# B&R Automation Studio project reAM250plc (part 2)

#### IOModule_X20AI4622.cpp
```cpp
/*++

Copyright (C) 2024 Institute for Machine Tools and Industrial Management
TUM School of Engineering and Design
Technical University of Munich

All rights reserved.

Redistribution and use in source and binary forms, with or without
modification, are permitted provided that the following conditions are met:
	* Redistributions of source code must retain the above copyright
	  notice, this list of conditions and the following disclaimer.
	* Redistributions in binary form must reproduce the above copyright
	  notice, this list of conditions and the following disclaimer in the
	  documentation and/or other materials provided with the distribution.
	* Neither the name of the Technical University of Munich nor the
	  names of its contributors may be used to endorse or promote products
	  derived from this software without specific prior written permission.

THIS SOFTWARE IS PROVIDED BY THE COPYRIGHT HOLDERS AND CONTRIBUTORS "AS IS" AND
ANY EXPRESS OR IMPLIED WARRANTIES, INCLUDING, BUT NOT LIMITED TO, THE IMPLIED
WARRANTIES OF MERCHANTABILITY AND FITNESS FOR A PARTICULAR PURPOSE ARE
DISCLAIMED. IN NO EVENT SHALL TECHNICAL UNIVERSITY OF MUNICH BE LIABLE FOR ANY
DIRECT, INDIRECT, INCIDENTAL, SPECIAL, EXEMPLARY, OR CONSEQUENTIAL DAMAGES
(INCLUDING, BUT NOT LIMITED TO, PROCUREMENT OF SUBSTITUTE GOODS OR SERVICES;
LOSS OF USE, DATA, OR PROFITS; OR BUSINESS INTERRUPTION) HOWEVER CAUSED AND
ON ANY THEORY OF LIABILITY, WHETHER IN CONTRACT, STRICT LIABILITY, OR TORT
(INCLUDING NEGLIGENCE OR OTHERWISE) ARISING IN ANY WAY OUT OF THE USE OF THIS
SOFTWARE, EVEN IF ADVISED OF THE POSSIBILITY OF SUCH DAMAGE.

*/

#include "IOModule_X20AI4622.hpp"

// Raw Registers
#define JOURNALVARIABLE_X20AI4622_MODULEOK 1
#define JOURNALVARIABLE_X20AI4622_STALEDATA 2
#define JOURNALVARIABLE_X20AI4622_SERIALNUMBER 3
#define JOURNALVARIABLE_X20AI4622_MODULEID 4
#define JOURNALVARIABLE_X20AI4622_HARDWAREVARIANT 5
#define JOURNALVARIABLE_X20AI4622_FIRMWAREVERSION 6
#define JOURNALVARIABLE_X20AI4622_ANALOGINPUT01 7
#define JOURNALVARIABLE_X20AI4622_ANALOGINPUT02 8
#define JOURNALVARIABLE_X20AI4622_ANALOGINPUT03 9
#define JOURNALVARIABLE_X20AI4622_ANALOGINPUT04 10
#define JOURNALVARIABLE_X20AI4622_STATUSINPUT01 11

// Derived Values
#define JOURNALVARIABLE_X20AI4622_INPUTVOLTAGE01 1001
#define JOURNALVARIABLE_X20AI4622_INPUTVOLTAGE02 1002
#define JOURNALVARIABLE_X20AI4622_INPUTVOLTAGE03 1003
#define JOURNALVARIABLE_X20AI4622_INPUTVOLTAGE04 1004
#define JOURNALVARIABLE_X20AI4622_INPUTCURRENTINAMPERE01 1005
#define JOURNALVARIABLE_X20AI4622_INPUTCURRENTINAMPERE02 1006
#define JOURNALVARIABLE_X20AI4622_INPUTCURRENTINAMPERE03 1007
#define JOURNALVARIABLE_X20AI4622_INPUTCURRENTINAMPERE04 1008

namespace BuRCPP {

	CIOModule_X20AI4622	::CIOModule_X20AI4622 (const std::string & sName, IOMappingX20AI4622_TYP * pMapping)
	: CIOModule (sName), m_pMapping (pMapping)
	{
		for (auto &channelType:m_ChannelTypes)
			channelType = eIOChannelType_X20AI4622::mtVoltage10V;

		for (auto &LowerLimits:m_nLowerLimit)
			LowerLimits = -32767;

		for (auto &UpperLimits:m_nUpperLimit)
			UpperLimits = 32766;

	}

	CIOModule_X20AI4622::~CIOModule_X20AI4622 ()
	{

	}

	void CIOModule_X20AI4622::onRegisterJournal ()
	{
		registerBoolValue ("ModuleOk", JOURNALVARIABLE_X20AI4622_MODULEOK);
		registerBoolValue ("StaleData", JOURNALVARIABLE_X20AI4622_STALEDATA);
		registerUInt32Value ("SerialNumber", JOURNALVARIABLE_X20AI4622_SERIALNUMBER);
		registerUInt16Value ("ModuleID", JOURNALVARIABLE_X20AI4622_MODULEID);
		registerUInt16Value ("HardwareVariant", JOURNALVARIABLE_X20AI4622_HARDWAREVARIANT);
		registerUInt16Value ("FirmwareVersion", JOURNALVARIABLE_X20AI4622_FIRMWAREVERSION);
		registerInt16Value ("AnalogInput01", JOURNALVARIABLE_X20AI4622_ANALOGINPUT01);
		registerInt16Value ("AnalogInput02", JOURNALVARIABLE_X20AI4622_ANALOGINPUT02);
		registerInt16Value ("AnalogInput03", JOURNALVARIABLE_X20AI4622_ANALOGINPUT03);
		registerInt16Value ("AnalogInput04", JOURNALVARIABLE_X20AI4622_ANALOGINPUT04);
		registerUInt8Value ("StatusInput01", JOURNALVARIABLE_X20AI4622_STATUSINPUT01);

		switch (getChannelType (1)) {
			case eIOChannelType_X20AI4622::mtVoltage10V:
				registerDoubleValue ("InputVoltage01", JOURNALVARIABLE_X20AI4622_INPUTVOLTAGE01, -10.0, 10.0, 65536);
				break;

			case eIOChannelType_X20AI4622::mtCurrent0to20mA:
				registerDoubleValue ("InputCurrentInAmpere01", JOURNALVARIABLE_X20AI4622_INPUTCURRENTINAMPERE01, 0.000, 0.020, 65536);
				break;

			case eIOChannelType_X20AI4622::mtCurrent4to20mA:
				registerDoubleValue ("InputCurrentInAmpere01", JOURNALVARIABLE_X20AI4622_INPUTCURRENTINAMPERE01, 0.004, 0.020, 65536);
				break;
		}

		switch (getChannelType (2)) {
			case eIOChannelType_X20AI4622::mtVoltage10V:
				registerDoubleValue ("InputVoltage02", JOURNALVARIABLE_X20AI4622_INPUTVOLTAGE02, -10.0, 10.0, 65536);
				break;

			case eIOChannelType_X20AI4622::mtCurrent0to20mA:
				registerDoubleValue ("InputCurrentInAmpere02", JOURNALVARIABLE_X20AI4622_INPUTCURRENTINAMPERE02, 0.000, 0.020, 65536);
				break;

			case eIOChannelType_X20AI4622::mtCurrent4to20mA:
				registerDoubleValue ("InputCurrentInAmpere02", JOURNALVARIABLE_X20AI4622_INPUTCURRENTINAMPERE02, 0.004, 0.020, 65536);
				break;
		}

		switch (getChannelType (3)) {
			case eIOChannelType_X20AI4622::mtVoltage10V:
				registerDoubleValue ("InputVoltage03", JOURNALVARIABLE_X20AI4622_INPUTVOLTAGE03, -10.0, 10.0, 65536);
				break;

			case eIOChannelType_X20AI4622::mtCurrent0to20mA:
				registerDoubleValue ("InputCurrentInAmpere03", JOURNALVARIABLE_X20AI4622_INPUTCURRENTINAMPERE03, 0.000, 0.020, 65536);
				break;

			case eIOChannelType_X20AI4622::mtCurrent4to20mA:
				registerDoubleValue ("InputCurrentInAmpere03", JOURNALVARIABLE_X20AI4622_INPUTCURRENTINAMPERE03, 0.004, 0.020, 65536);
				break;
		}

		switch (getChannelType (4)) {
			case eIOChannelType_X20AI4622::mtVoltage10V:
				registerDoubleValue ("InputVoltage04", JOURNALVARIABLE_X20AI4622_INPUTVOLTAGE04, -10.0, 10.0, 65536);
				break;

			case eIOChannelType_X20AI4622::mtCurrent0to20mA:
				registerDoubleValue ("InputCurrentInAmpere04", JOURNALVARIABLE_X20AI4622_INPUTCURRENTINAMPERE04, 0.000, 0.020, 65536);
				break;

			case eIOChannelType_X20AI4622::mtCurrent4to20mA:
				registerDoubleValue ("InputCurrentInAmpere04", JOURNALVARIABLE_X20AI4622_INPUTCURRENTINAMPERE04, 0.004, 0.020, 65536);
				break;
		}
	}

	void CIOModule_X20AI4622::onUpdateJournal ()
	{
		setBoolValue (JOURNALVARIABLE_X20AI4622_MODULEOK, m_pMapping->ModuleOk);
		setBoolValue (JOURNALVARIABLE_X20AI4622_STALEDATA, m_pMapping->StaleData);
		setIntegerValue (JOURNALVARIABLE_X20AI4622_SERIALNUMBER, m_pMapping->SerialNumber);
		setIntegerValue (JOURNALVARIABLE_X20AI4622_MODULEID, m_pMapping->ModuleID);
		setIntegerValue (JOURNALVARIABLE_X20AI4622_HARDWAREVARIANT, m_pMapping->HardwareVariant);
		setIntegerValue (JOURNALVARIABLE_X20AI4622_FIRMWAREVERSION, m_pMapping->FirmwareVersion);
		setIntegerValue (JOURNALVARIABLE_X20AI4622_ANALOGINPUT01, m_pMapping->AnalogInput01);
		setIntegerValue (JOURNALVARIABLE_X20AI4622_ANALOGINPUT02, m_pMapping->AnalogInput02);
		setIntegerValue (JOURNALVARIABLE_X20AI4622_ANALOGINPUT03, m_pMapping->AnalogInput03);
		setIntegerValue (JOURNALVARIABLE_X20AI4622_ANALOGINPUT04, m_pMapping->AnalogInput04);
		setIntegerValue (JOURNALVARIABLE_X20AI4622_STATUSINPUT01, m_pMapping->StatusInput01);

		for (int index = 0; index < 4; index++)
		{
			uint32_t nChannelNo = index + 1;
			switch (getChannelType (nChannelNo)) {

				case eIOChannelType_X20AI4622::mtVoltage10V:

					setDoubleValue (JOURNALVARIABLE_X20AI4622_INPUTVOLTAGE01 + index, getInputVoltageInVolt (nChannelNo));
					/*setDoubleValue (JOURNALVARIABLE_X20AI4622_INPUTVOLTAGE02, getInputVoltageInVolt (2));
					setDoubleValue (JOURNALVARIABLE_X20AI4622_INPUTVOLTAGE03, getInputVoltageInVolt (3));
					setDoubleValue (JOURNALVARIABLE_X20AI4622_INPUTVOLTAGE04, getInputVoltageInVolt (4));*/
					break;

				case eIOChannelType_X20AI4622::mtCurrent0to20mA:
				case eIOChannelType_X20AI4622::mtCurrent4to20mA:
					setDoubleValue (JOURNALVARIABLE_X20AI4622_INPUTCURRENTINAMPERE01 + index, getInputCurrentInAmpere (nChannelNo));
					/*setDoubleValue (JOURNALVARIABLE_X20AI4622_INPUTCURRENTINAMPERE02, getInputCurrentInAmpere (2));
					setDoubleValue (JOURNALVARIABLE_X20AI4622_INPUTCURRENTINAMPERE03, getInputCurrentInAmpere (3));
					setDoubleValue (JOURNALVARIABLE_X20AI4622_INPUTCURRENTINAMPERE04, getInputCurrentInAmpere (4));*/
					break;
			}
		}
	}

	bool CIOModule_X20AI4622::isActive ()
	{
		return m_pMapping->ModuleOk != 0;
	}

	uint32_t CIOModule_X20AI4622::getSerialNumber ()
	{
		return m_pMapping->SerialNumber;
	}

	uint16_t CIOModule_X20AI4622::getModuleID ()
	{
		return m_pMapping->ModuleID;
	}

	uint16_t CIOModule_X20AI4622::getHardwareVariant ()
	{
		return m_pMapping->HardwareVariant;
	}

	uint16_t CIOModule_X20AI4622::getFirmwareVersion ()
	{
		return m_pMapping->FirmwareVersion;
	}

	int16_t CIOModule_X20AI4622::getRawValue (uint32_t nChannelNo)
	{

		switch (nChannelNo) {
			case 1: return m_pMapping->AnalogInput01;
			case 2: return m_pMapping->AnalogInput02;
			case 3: return m_pMapping->AnalogInput03;
			case 4: return m_pMapping->AnalogInput04;
			default:
				throw CException (eErrorCode::INVALIDCHANNELNUMBER, "invalid channel number: " + std::to_string (nChannelNo));
		}
	}

	double CIOModule_X20AI4622::getRawValueNormalizedZeroToOne (uint32_t nChannelNo)
	{
		if (nChannelNo > 0 && nChannelNo < 5)
		{
			int32_t rawValue = getRawValue (nChannelNo);
			int32_t nRange = m_nUpperLimit[nChannelNo -1] - m_nLowerLimit[nChannelNo -1];
			return (double) (rawValue - (int32_t) m_nLowerLimit[nChannelNo -1]) / (double) nRange;
		}
		else
		{
			throw CException (eErrorCode::INVALIDCHANNELNUMBER, "invalid channel number: " + std::to_string (nChannelNo));
		}
	}

	double CIOModule_X20AI4622::getInputVoltageInVolt (uint32_t nChannelNo)
	{
		switch (getChannelType (nChannelNo)) {
			case eIOChannelType_X20AI4622::mtVoltage10V:
				return (getRawValueNormalizedZeroToOne (nChannelNo) - 0.5) * 20.0;
			default:
				throw CException (eErrorCode::NOVOLTAGEMODULE, "IO module does not measure voltage: " + m_sName );
		}

	}

	double CIOModule_X20AI4622::getInputCurrentInAmpere (uint32_t nChannelNo)
	{
		switch (getChannelType (nChannelNo)) {
			case eIOChannelType_X20AI4622::mtCurrent0to20mA:
				return (getRawValueNormalizedZeroToOne (nChannelNo)) * 0.020;
			case eIOChannelType_X20AI4622::mtCurrent4to20mA:
				return (getRawValueNormalizedZeroToOne (nChannelNo)) * 0.016 + 0.004;
			default:
				throw CException (eErrorCode::NOCURRENTMODULE, "IO module does not measure current: " + m_sName );
		}

	}

	bool CIOModule_X20AI4622::setRange(uint32_t nChannelNo, uint16_t nLower, uint16_t nUpper)
	{
		if (nChannelNo > 0 && nChannelNo < 5)
		{
			m_nLowerLimit[nChannelNo - 1] = nLower;
			m_nUpperLimit[nChannelNo - 1] = nUpper;
			return true;
		}
		else
		{
			return false;
		}
	}

	uint16_t CIOModule_X20AI4622::getIOStatus (uint32_t nChannelNo)
	{
		//status IDs: 0 = no error, 1 = lower limit value undershot, 2 = upper limit value exceeded, 3 = wire breakage
		switch (nChannelNo) {
			case 1: return (m_pMapping->StatusInput01 & 0x03);
			case 2: return ((m_pMapping->StatusInput01 >> 2) & 0x03);
			case 3: return ((m_pMapping->StatusInput01 >> 4) & 0x03);
			case 4: return ((m_pMapping->StatusInput01 >> 6) & 0x03);
			default:
				throw CException (eErrorCode::INVALIDCHANNELNUMBER, "invalid channel number: " + std::to_string (nChannelNo));
		}
	}

	eIOChannelType_X20AI4622 CIOModule_X20AI4622::getChannelType (uint32_t nChannelNo)
	{
		if ((nChannelNo >= 1) && (nChannelNo <= 4))
		{
			return m_ChannelTypes[nChannelNo - 1];
		}
		else
			return eIOChannelType_X20AI4622::mtUnknown;
	}

	bool CIOModule_X20AI4622::setChannelType (uint32_t nChannelNo, eIOChannelType_X20AI4622 eChannelTypes)
	{
		if ((nChannelNo >= 1) && (nChannelNo <= 4))
		{
			switch (eChannelTypes) {
				case eIOChannelType_X20AI4622::mtVoltage10V:
					setRange(nChannelNo, -32768 , 32767);
					break;
				case eIOChannelType_X20AI4622::mtCurrent0to20mA:
					setRange(nChannelNo, 0, 32767);
					break;
				case eIOChannelType_X20AI4622::mtCurrent4to20mA:
					setRange(nChannelNo, -8192 , 32767);
					break;
				default:
					throw CException (eErrorCode::INVALIDCHANNELTYPE, "invalid channel type");
			}
			m_ChannelTypes[nChannelNo - 1] = eChannelTypes;
			return true;
		}
		else
		{
			throw CException (eErrorCode::INVALIDCHANNELNUMBER, "invalid channel number: " + std::to_string (nChannelNo));
		}
	}

}
```

#### IOModule_X20DI6371.hpp
```cpp
/*++

Copyright (C) 2024 Institute for Machine Tools and Industrial Management
TUM School of Engineering and Design
Technical University of Munich

All rights reserved.

Redistribution and use in source and binary forms, with or without
modification, are permitted provided that the following conditions are met:
	* Redistributions of source code must retain the above copyright
	  notice, this list of conditions and the following disclaimer.
	* Redistributions in binary form must reproduce the above copyright
	  notice, this list of conditions and the following disclaimer in the
	  documentation and/or other materials provided with the distribution.
	* Neither the name of the Technical University of Munich nor the
	  names of its contributors may be used to endorse or promote products
	  derived from this software without specific prior written permission.

THIS SOFTWARE IS PROVIDED BY THE COPYRIGHT HOLDERS AND CONTRIBUTORS "AS IS" AND
ANY EXPRESS OR IMPLIED WARRANTIES, INCLUDING, BUT NOT LIMITED TO, THE IMPLIED
WARRANTIES OF MERCHANTABILITY AND FITNESS FOR A PARTICULAR PURPOSE ARE
DISCLAIMED. IN NO EVENT SHALL TECHNICAL UNIVERSITY OF MUNICH BE LIABLE FOR ANY
DIRECT, INDIRECT, INCIDENTAL, SPECIAL, EXEMPLARY, OR CONSEQUENTIAL DAMAGES
(INCLUDING, BUT NOT LIMITED TO, PROCUREMENT OF SUBSTITUTE GOODS OR SERVICES;
LOSS OF USE, DATA, OR PROFITS; OR BUSINESS INTERRUPTION) HOWEVER CAUSED AND
ON ANY THEORY OF LIABILITY, WHETHER IN CONTRACT, STRICT LIABILITY, OR TORT
(INCLUDING NEGLIGENCE OR OTHERWISE) ARISING IN ANY WAY OUT OF THE USE OF THIS
SOFTWARE, EVEN IF ADVISED OF THE POSSIBILITY OF SUCH DAMAGE.

*/

#ifndef __IOMODULE_X20DI6371_HPP
#define __IOMODULE_X20DI6371_HPP

#include "../Framework/Framework.hpp"

namespace BuRCPP {

	class CIOModule_X20DI6371 : public CIOModule {
		protected:
		IOMappingX20DI6371_TYP * m_pMapping;

		public:
		CIOModule_X20DI6371 (const std::string & sName, IOMappingX20DI6371_TYP * pMapping);
		virtual ~CIOModule_X20DI6371 ();

		bool isActive () override;
		uint32_t getSerialNumber () override;
		uint16_t getModuleID () override;
		uint16_t getHardwareVariant () override;
		uint16_t getFirmwareVersion () override;

		uint16_t getInput (uint32_t);

		void onRegisterJournal ();
		void onUpdateJournal ();

	};

}

#endif // __IOMODULE_X20DI6371_HPP
```

#### IOModule_X20DI6371.cpp
```cpp
/*++

Copyright (C) 2024 Institute for Machine Tools and Industrial Management
TUM School of Engineering and Design
Technical University of Munich

All rights reserved.

Redistribution and use in source and binary forms, with or without
modification, are permitted provided that the following conditions are met:
	* Redistributions of source code must retain the above copyright
	  notice, this list of conditions and the following disclaimer.
	* Redistributions in binary form must reproduce the above copyright
	  notice, this list of conditions and the following disclaimer in the
	  documentation and/or other materials provided with the distribution.
	* Neither the name of the Technical University of Munich nor the
	  names of its contributors may be used to endorse or promote products
	  derived from this software without specific prior written permission.

THIS SOFTWARE IS PROVIDED BY THE COPYRIGHT HOLDERS AND CONTRIBUTORS "AS IS" AND
ANY EXPRESS OR IMPLIED WARRANTIES, INCLUDING, BUT NOT LIMITED TO, THE IMPLIED
WARRANTIES OF MERCHANTABILITY AND FITNESS FOR A PARTICULAR PURPOSE ARE
DISCLAIMED. IN NO EVENT SHALL TECHNICAL UNIVERSITY OF MUNICH BE LIABLE FOR ANY
DIRECT, INDIRECT, INCIDENTAL, SPECIAL, EXEMPLARY, OR CONSEQUENTIAL DAMAGES
(INCLUDING, BUT NOT LIMITED TO, PROCUREMENT OF SUBSTITUTE GOODS OR SERVICES;
LOSS OF USE, DATA, OR PROFITS; OR BUSINESS INTERRUPTION) HOWEVER CAUSED AND
ON ANY THEORY OF LIABILITY, WHETHER IN CONTRACT, STRICT LIABILITY, OR TORT
(INCLUDING NEGLIGENCE OR OTHERWISE) ARISING IN ANY WAY OUT OF THE USE OF THIS
SOFTWARE, EVEN IF ADVISED OF THE POSSIBILITY OF SUCH DAMAGE.

*/

#include "IOModule_X20DI6371.hpp"

// Raw Registers
#define JOURNALVARIABLE_X20DI6371_MODULEOK 1
#define JOURNALVARIABLE_X20DI6371_SERIALNUMBER 2
#define JOURNALVARIABLE_X20DI6371_MODULEID 3
#define JOURNALVARIABLE_X20DI6371_HARDWAREVARIANT 4
#define JOURNALVARIABLE_X20DI6371_FIRMWAREVERSION 5
#define JOURNALVARIABLE_X20DI6371_DIGITALINPUT01 6
#define JOURNALVARIABLE_X20DI6371_DIGITALINPUT02 7
#define JOURNALVARIABLE_X20DI6371_DIGITALINPUT03 8
#define JOURNALVARIABLE_X20DI6371_DIGITALINPUT04 9
#define JOURNALVARIABLE_X20DI6371_DIGITALINPUT05 10
#define JOURNALVARIABLE_X20DI6371_DIGITALINPUT06 11

namespace BuRCPP {

	CIOModule_X20DI6371::CIOModule_X20DI6371 (const std::string & sName, IOMappingX20DI6371_TYP * pMapping)
		: CIOModule (sName), m_pMapping (pMapping)
	{

	}

	CIOModule_X20DI6371::~CIOModule_X20DI6371 ()
	{
	}

	void CIOModule_X20DI6371::onRegisterJournal ()
	{
		registerBoolValue ("ModuleOk", JOURNALVARIABLE_X20DI6371_MODULEOK);
		registerUInt32Value ("SerialNumber", JOURNALVARIABLE_X20DI6371_SERIALNUMBER);
		registerUInt16Value ("ModuleID", JOURNALVARIABLE_X20DI6371_MODULEID);
		registerUInt16Value ("HardwareVariant", JOURNALVARIABLE_X20DI6371_HARDWAREVARIANT);
		registerUInt16Value ("FirmwareVersion", JOURNALVARIABLE_X20DI6371_FIRMWAREVERSION);
		registerBoolValue ("DigitalInput01", JOURNALVARIABLE_X20DI6371_DIGITALINPUT01);
		registerBoolValue ("DigitalInput02", JOURNALVARIABLE_X20DI6371_DIGITALINPUT02);
		registerBoolValue ("DigitalInput03", JOURNALVARIABLE_X20DI6371_DIGITALINPUT03);
		registerBoolValue ("DigitalInput04", JOURNALVARIABLE_X20DI6371_DIGITALINPUT04);
		registerBoolValue ("DigitalInput05", JOURNALVARIABLE_X20DI6371_DIGITALINPUT05);
		registerBoolValue ("DigitalInput06", JOURNALVARIABLE_X20DI6371_DIGITALINPUT06);

	}

	void CIOModule_X20DI6371::onUpdateJournal ()
	{
		setBoolValue (JOURNALVARIABLE_X20DI6371_MODULEOK, m_pMapping->ModuleOk);
		setIntegerValue (JOURNALVARIABLE_X20DI6371_SERIALNUMBER, m_pMapping->SerialNumber);
		setIntegerValue (JOURNALVARIABLE_X20DI6371_MODULEID, m_pMapping->ModuleID);
		setIntegerValue (JOURNALVARIABLE_X20DI6371_HARDWAREVARIANT, m_pMapping->HardwareVariant);
		setIntegerValue (JOURNALVARIABLE_X20DI6371_FIRMWAREVERSION, m_pMapping->FirmwareVersion);
		setBoolValue (JOURNALVARIABLE_X20DI6371_DIGITALINPUT01, m_pMapping->DigitalInput01);
		setBoolValue (JOURNALVARIABLE_X20DI6371_DIGITALINPUT02, m_pMapping->DigitalInput02);
		setBoolValue (JOURNALVARIABLE_X20DI6371_DIGITALINPUT03, m_pMapping->DigitalInput03);
		setBoolValue (JOURNALVARIABLE_X20DI6371_DIGITALINPUT04, m_pMapping->DigitalInput04);
		setBoolValue (JOURNALVARIABLE_X20DI6371_DIGITALINPUT05, m_pMapping->DigitalInput05);
		setBoolValue (JOURNALVARIABLE_X20DI6371_DIGITALINPUT06, m_pMapping->DigitalInput06);
	}

	bool CIOModule_X20DI6371::isActive ()
	{
		return m_pMapping->ModuleOk != 0;
	}

	uint32_t CIOModule_X20DI6371::getSerialNumber ()
	{
		return m_pMapping->SerialNumber;
	}

	uint16_t CIOModule_X20DI6371::getModuleID ()
	{
		return m_pMapping->ModuleID;
	}

	uint16_t CIOModule_X20DI6371::getHardwareVariant ()
	{
		return m_pMapping->HardwareVariant;
	}

	uint16_t CIOModule_X20DI6371::getFirmwareVersion ()
	{
		return m_pMapping->FirmwareVersion;
	}

	uint16_t CIOModule_X20DI6371::getInput (uint32_t nChannelNo)
	{
		switch (nChannelNo)
		{
			case 1:
				return m_pMapping->DigitalInput01;
				break;

			case 2:
				return m_pMapping->DigitalInput02;
				break;

			case 3:
				return m_pMapping->DigitalInput03;
				break;

			case 4:
				return m_pMapping->DigitalInput04;
				break;

			case 5:
				return m_pMapping->DigitalInput05;
				break;

			case 6:
				return m_pMapping->DigitalInput06;
				break;
			default:
				return 0;
				break;

		}
	}

}
```

#### IOModule_X20DI9371.hpp
```cpp
/*++

Copyright (C) 2024 Institute for Machine Tools and Industrial Management
TUM School of Engineering and Design
Technical University of Munich

All rights reserved.

Redistribution and use in source and binary forms, with or without
modification, are permitted provided that the following conditions are met:
	* Redistributions of source code must retain the above copyright
	  notice, this list of conditions and the following disclaimer.
	* Redistributions in binary form must reproduce the above copyright
	  notice, this list of conditions and the following disclaimer in the
	  documentation and/or other materials provided with the distribution.
	* Neither the name of the Technical University of Munich nor the
	  names of its contributors may be used to endorse or promote products
	  derived from this software without specific prior written permission.

THIS SOFTWARE IS PROVIDED BY THE COPYRIGHT HOLDERS AND CONTRIBUTORS "AS IS" AND
ANY EXPRESS OR IMPLIED WARRANTIES, INCLUDING, BUT NOT LIMITED TO, THE IMPLIED
WARRANTIES OF MERCHANTABILITY AND FITNESS FOR A PARTICULAR PURPOSE ARE
DISCLAIMED. IN NO EVENT SHALL TECHNICAL UNIVERSITY OF MUNICH BE LIABLE FOR ANY
DIRECT, INDIRECT, INCIDENTAL, SPECIAL, EXEMPLARY, OR CONSEQUENTIAL DAMAGES
(INCLUDING, BUT NOT LIMITED TO, PROCUREMENT OF SUBSTITUTE GOODS OR SERVICES;
LOSS OF USE, DATA, OR PROFITS; OR BUSINESS INTERRUPTION) HOWEVER CAUSED AND
ON ANY THEORY OF LIABILITY, WHETHER IN CONTRACT, STRICT LIABILITY, OR TORT
(INCLUDING NEGLIGENCE OR OTHERWISE) ARISING IN ANY WAY OUT OF THE USE OF THIS
SOFTWARE, EVEN IF ADVISED OF THE POSSIBILITY OF SUCH DAMAGE.

*/

#ifndef __IOMODULE_X20DI9371_HPP
#define __IOMODULE_X20DI9371_HPP

#include "../Framework/Framework.hpp"

namespace BuRCPP {

	class CIOModule_X20DI9371 : public CIOModule {
		protected:
		IOMappingX20DI9371_TYP * m_pMapping;

		public:
		CIOModule_X20DI9371 (const std::string & sName, IOMappingX20DI9371_TYP * pMapping);
		virtual ~CIOModule_X20DI9371 ();

		bool isActive () override;
		uint32_t getSerialNumber () override;
		uint16_t getModuleID () override;
		uint16_t getHardwareVariant () override;
		uint16_t getFirmwareVersion () override;

		bool getChannelValue (uint32_t nChannelNo);

	};

}

#endif // __IOMODULE_X20DI9371_HPP
```

#### IOModule_X20DI9371.cpp
```cpp
/*++

Copyright (C) 2024 Institute for Machine Tools and Industrial Management
TUM School of Engineering and Design
Technical University of Munich

All rights reserved.

Redistribution and use in source and binary forms, with or without
modification, are permitted provided that the following conditions are met:
	* Redistributions of source code must retain the above copyright
	  notice, this list of conditions and the following disclaimer.
	* Redistributions in binary form must reproduce the above copyright
	  notice, this list of conditions and the following disclaimer in the
	  documentation and/or other materials provided with the distribution.
	* Neither the name of the Technical University of Munich nor the
	  names of its contributors may be used to endorse or promote products
	  derived from this software without specific prior written permission.

THIS SOFTWARE IS PROVIDED BY THE COPYRIGHT HOLDERS AND CONTRIBUTORS "AS IS" AND
ANY EXPRESS OR IMPLIED WARRANTIES, INCLUDING, BUT NOT LIMITED TO, THE IMPLIED
WARRANTIES OF MERCHANTABILITY AND FITNESS FOR A PARTICULAR PURPOSE ARE
DISCLAIMED. IN NO EVENT SHALL TECHNICAL UNIVERSITY OF MUNICH BE LIABLE FOR ANY
DIRECT, INDIRECT, INCIDENTAL, SPECIAL, EXEMPLARY, OR CONSEQUENTIAL DAMAGES
(INCLUDING, BUT NOT LIMITED TO, PROCUREMENT OF SUBSTITUTE GOODS OR SERVICES;
LOSS OF USE, DATA, OR PROFITS; OR BUSINESS INTERRUPTION) HOWEVER CAUSED AND
ON ANY THEORY OF LIABILITY, WHETHER IN CONTRACT, STRICT LIABILITY, OR TORT
(INCLUDING NEGLIGENCE OR OTHERWISE) ARISING IN ANY WAY OUT OF THE USE OF THIS
SOFTWARE, EVEN IF ADVISED OF THE POSSIBILITY OF SUCH DAMAGE.

*/
```

#### IOModule_X20SI8110.cpp
```cpp
/*++

Copyright (C) 2024 Institute for Machine Tools and Industrial Management
TUM School of Engineering and Design
Technical University of Munich

All rights reserved.

Redistribution and use in source and binary forms, with or without
modification, are permitted provided that the following conditions are met:
	* Redistributions of source code must retain the above copyright
	  notice, this list of conditions and the following disclaimer.
	* Redistributions in binary form must reproduce the above copyright
	  notice, this list of conditions and the following disclaimer in the
	  documentation and/or other materials provided with the distribution.
	* Neither the name of the Technical University of Munich nor the
	  names of its contributors may be used to endorse or promote products
	  derived from this software without specific prior written permission.

THIS SOFTWARE IS PROVIDED BY THE COPYRIGHT HOLDERS AND CONTRIBUTORS "AS IS" AND
ANY EXPRESS OR IMPLIED WARRANTIES, INCLUDING, BUT NOT LIMITED TO, THE IMPLIED
WARRANTIES OF MERCHANTABILITY AND FITNESS FOR A PARTICULAR PURPOSE ARE
DISCLAIMED. IN NO EVENT SHALL TECHNICAL UNIVERSITY OF MUNICH BE LIABLE FOR ANY
DIRECT, INDIRECT, INCIDENTAL, SPECIAL, EXEMPLARY, OR CONSEQUENTIAL DAMAGES
(INCLUDING, BUT NOT LIMITED TO, PROCUREMENT OF SUBSTITUTE GOODS OR SERVICES;
LOSS OF USE, DATA, OR PROFITS; OR BUSINESS INTERRUPTION) HOWEVER CAUSED AND
ON ANY THEORY OF LIABILITY, WHETHER IN CONTRACT, STRICT LIABILITY, OR TORT
(INCLUDING NEGLIGENCE OR OTHERWISE) ARISING IN ANY WAY OUT OF THE USE OF THIS
SOFTWARE, EVEN IF ADVISED OF THE POSSIBILITY OF SUCH DAMAGE.

*/

#include "IOModule_X20SI8110.hpp"

// Raw Registers
#define JOURNALVARIABLE_X20SI8110_MODULEOK 1
#define JOURNALVARIABLE_X20SI8110_SERIALNUMBER 2
#define JOURNALVARIABLE_X20SI8110_MODULEID 3
#define JOURNALVARIABLE_X20SI8110_HARDWAREVARIANT 4
#define JOURNALVARIABLE_X20SI8110_FIRMWAREVERSION 5
#define JOURNALVARIABLE_X20SI8110_SAFEMODULEOK 6
#define JOURNALVARIABLE_X20SI8110_SAFEDIGITALINPUT01 7
#define JOURNALVARIABLE_X20SI8110_SAFEDIGITALINPUT02 8
#define JOURNALVARIABLE_X20SI8110_SAFEDIGITALINPUT03 9
#define JOURNALVARIABLE_X20SI8110_SAFEDIGITALINPUT04 10
#define JOURNALVARIABLE_X20SI8110_SAFEDIGITALINPUT05 11
#define JOURNALVARIABLE_X20SI8110_SAFEDIGITALINPUT06 12
#define JOURNALVARIABLE_X20SI8110_SAFEDIGITALINPUT07 13
#define JOURNALVARIABLE_X20SI8110_SAFEDIGITALINPUT08 14
#define JOURNALVARIABLE_X20SI8110_SAFETWOCHANNELINPUT0102 15
#define JOURNALVARIABLE_X20SI8110_SAFETWOCHANNELINPUT0304 16
#define JOURNALVARIABLE_X20SI8110_SAFETWOCHANNELINPUT0506 17
#define JOURNALVARIABLE_X20SI8110_SAFETWOCHANNELINPUT0708 18
#define JOURNALVARIABLE_X20SI8110_SAFEINPUTOK01 19
#define JOURNALVARIABLE_X20SI8110_SAFEINPUTOK02 20
#define JOURNALVARIABLE_X20SI8110_SAFEINPUTOK03 21
#define JOURNALVARIABLE_X20SI8110_SAFEINPUTOK04 22
#define JOURNALVARIABLE_X20SI8110_SAFEINPUTOK05 23
#define JOURNALVARIABLE_X20SI8110_SAFEINPUTOK06 24
#define JOURNALVARIABLE_X20SI8110_SAFEINPUTOK07 25
#define JOURNALVARIABLE_X20SI8110_SAFEINPUTOK08 26
#define JOURNALVARIABLE_X20SI8110_SAFETWOCHANNELOK0102 27
#define JOURNALVARIABLE_X20SI8110_SAFETWOCHANNELOK0304 28
#define JOURNALVARIABLE_X20SI8110_SAFETWOCHANNELOK0506 29
#define JOURNALVARIABLE_X20SI8110_SAFETWOCHANNELOK0708 30

namespace BuRCPP {

	CIOModule_X20SI8110::CIOModule_X20SI8110 (const std::string & sName, IOMappingX20SI8110_TYP * pMapping)
		: CIOModule (sName), m_pMapping (pMapping)
	{

	}

	CIOModule_X20SI8110::~CIOModule_X20SI8110 ()
	{
	}

	void CIOModule_X20SI8110::onRegisterJournal ()
	{
		registerBoolValue ("ModuleOk", JOURNALVARIABLE_X20SI8110_MODULEOK);
		registerUInt32Value ("SerialNumber", JOURNALVARIABLE_X20SI8110_SERIALNUMBER);
		registerUInt16Value ("ModuleID", JOURNALVARIABLE_X20SI8110_MODULEID);
		registerUInt16Value ("HardwareVariant", JOURNALVARIABLE_X20SI8110_HARDWAREVARIANT);
		registerUInt16Value ("FirmwareVersion", JOURNALVARIABLE_X20SI8110_FIRMWAREVERSION);
		registerBoolValue ("SafeModuleOK", JOURNALVARIABLE_X20SI8110_SAFEMODULEOK);
		registerBoolValue ("SafeDigitalInput01", JOURNALVARIABLE_X20SI8110_SAFEDIGITALINPUT01);
		registerBoolValue ("SafeDigitalInput02", JOURNALVARIABLE_X20SI8110_SAFEDIGITALINPUT02);
		registerBoolValue ("SafeDigitalInput03", JOURNALVARIABLE_X20SI8110_SAFEDIGITALINPUT03);
		registerBoolValue ("SafeDigitalInput04", JOURNALVARIABLE_X20SI8110_SAFEDIGITALINPUT04);
		registerBoolValue ("SafeDigitalInput05", JOURNALVARIABLE_X20SI8110_SAFEDIGITALINPUT05);
		registerBoolValue ("SafeDigitalInput06", JOURNALVARIABLE_X20SI8110_SAFEDIGITALINPUT06);
		registerBoolValue ("SafeDigitalInput07", JOURNALVARIABLE_X20SI8110_SAFEDIGITALINPUT07);
		registerBoolValue ("SafeDigitalInput08", JOURNALVARIABLE_X20SI8110_SAFEDIGITALINPUT08);
		registerBoolValue ("SafeTwoChannelInput0102", JOURNALVARIABLE_X20SI8110_SAFETWOCHANNELINPUT0102);
		registerBoolValue ("SafeTwoChannelInput0304", JOURNALVARIABLE_X20SI8110_SAFETWOCHANNELINPUT0304);
		registerBoolValue ("SafeTwoChannelInput0506", JOURNALVARIABLE_X20SI8110_SAFETWOCHANNELINPUT0506);
		registerBoolValue ("SafeTwoChannelInput0708", JOURNALVARIABLE_X20SI8110_SAFETWOCHANNELINPUT0708);
		registerBoolValue ("SafeInputOK01", JOURNALVARIABLE_X20SI8110_SAFEINPUTOK01);
		registerBoolValue ("SafeInputOK02", JOURNALVARIABLE_X20SI8110_SAFEINPUTOK02);
		registerBoolValue ("SafeInputOK03", JOURNALVARIABLE_X20SI8110_SAFEINPUTOK03);
		registerBoolValue ("SafeInputOK04", JOURNALVARIABLE_X20SI8110_SAFEINPUTOK04);
		registerBoolValue ("SafeInputOK05", JOURNALVARIABLE_X20SI8110_SAFEINPUTOK05);
		registerBoolValue ("SafeInputOK06", JOURNALVARIABLE_X20SI8110_SAFEINPUTOK06);
		registerBoolValue ("SafeInputOK07", JOURNALVARIABLE_X20SI8110_SAFEINPUTOK07);
		registerBoolValue ("SafeInputOK08", JOURNALVARIABLE_X20SI8110_SAFEINPUTOK08);
		registerBoolValue ("SafeTwoChannelOK0102", JOURNALVARIABLE_X20SI8110_SAFETWOCHANNELOK0102);
		registerBoolValue ("SafeTwoChannelOK0304", JOURNALVARIABLE_X20SI8110_SAFETWOCHANNELOK0304);
		registerBoolValue ("SafeTwoChannelOK0506", JOURNALVARIABLE_X20SI8110_SAFETWOCHANNELOK0506);
		registerBoolValue ("SafeTwoChannelOK0708", JOURNALVARIABLE_X20SI8110_SAFETWOCHANNELOK0708);
	}

	void CIOModule_X20SI8110::onUpdateJournal ()
	{
		setBoolValue (JOURNALVARIABLE_X20SI8110_MODULEOK, m_pMapping->ModuleOk);
		setIntegerValue (JOURNALVARIABLE_X20SI8110_SERIALNUMBER, m_pMapping->SerialNumber);
		setIntegerValue (JOURNALVARIABLE_X20SI8110_MODULEID, m_pMapping->ModuleID);
		setIntegerValue (JOURNALVARIABLE_X20SI8110_HARDWAREVARIANT, m_pMapping->HardwareVariant);
		setIntegerValue (JOURNALVARIABLE_X20SI8110_FIRMWAREVERSION, m_pMapping->FirmwareVersion);
		setBoolValue (JOURNALVARIABLE_X20SI8110_SAFEMODULEOK, m_pMapping->SafeModuleOK);
		setBoolValue (JOURNALVARIABLE_X20SI8110_SAFEDIGITALINPUT01, m_pMapping->SafeDigitalInput01);
		setBoolValue (JOURNALVARIABLE_X20SI8110_SAFEDIGITALINPUT02, m_pMapping->SafeDigitalInput02);
		setBoolValue (JOURNALVARIABLE_X20SI8110_SAFEDIGITALINPUT03, m_pMapping->SafeDigitalInput03);
		setBoolValue (JOURNALVARIABLE_X20SI8110_SAFEDIGITALINPUT04, m_pMapping->SafeDigitalInput04);
		setBoolValue (JOURNALVARIABLE_X20SI8110_SAFEDIGITALINPUT05, m_pMapping->SafeDigitalInput05);
		setBoolValue (JOURNALVARIABLE_X20SI8110_SAFEDIGITALINPUT06, m_pMapping->SafeDigitalInput06);
		setBoolValue (JOURNALVARIABLE_X20SI8110_SAFEDIGITALINPUT07, m_pMapping->SafeDigitalInput07);
		setBoolValue (JOURNALVARIABLE_X20SI8110_SAFEDIGITALINPUT08, m_pMapping->SafeDigitalInput08);
		setBoolValue (JOURNALVARIABLE_X20SI8110_SAFETWOCHANNELINPUT0102, m_pMapping->SafeTwoChannelInput0102);
		setBoolValue (JOURNALVARIABLE_X20SI8110_SAFETWOCHANNELINPUT0304, m_pMapping->SafeTwoChannelInput0304);
		setBoolValue (JOURNALVARIABLE_X20SI8110_SAFETWOCHANNELINPUT0506, m_pMapping->SafeTwoChannelInput0506);
		setBoolValue (JOURNALVARIABLE_X20SI8110_SAFETWOCHANNELINPUT0708, m_pMapping->SafeTwoChannelInput0708);
		setBoolValue (JOURNALVARIABLE_X20SI8110_SAFEINPUTOK01, m_pMapping->SafeInputOK01);
		setBoolValue (JOURNALVARIABLE_X20SI8110_SAFEINPUTOK02, m_pMapping->SafeInputOK02);
		setBoolValue (JOURNALVARIABLE_X20SI8110_SAFEINPUTOK03, m_pMapping->SafeInputOK03);
		setBoolValue (JOURNALVARIABLE_X20SI8110_SAFEINPUTOK04, m_pMapping->SafeInputOK04);
		setBoolValue (JOURNALVARIABLE_X20SI8110_SAFEINPUTOK05, m_pMapping->SafeInputOK05);
		setBoolValue (JOURNALVARIABLE_X20SI8110_SAFEINPUTOK06, m_pMapping->SafeInputOK06);
		setBoolValue (JOURNALVARIABLE_X20SI8110_SAFEINPUTOK07, m_pMapping->SafeInputOK07);
		setBoolValue (JOURNALVARIABLE_X20SI8110_SAFEINPUTOK08, m_pMapping->SafeInputOK08);
		setBoolValue (JOURNALVARIABLE_X20SI8110_SAFETWOCHANNELOK0102, m_pMapping->SafeTwoChannelOK0102);
		setBoolValue (JOURNALVARIABLE_X20SI8110_SAFETWOCHANNELOK0304, m_pMapping->SafeTwoChannelOK0304);
		setBoolValue (JOURNALVARIABLE_X20SI8110_SAFETWOCHANNELOK0506, m_pMapping->SafeTwoChannelOK0506);
		setBoolValue (JOURNALVARIABLE_X20SI8110_SAFETWOCHANNELOK0708, m_pMapping->SafeTwoChannelOK0708);
	}

	bool CIOModule_X20SI8110::isActive ()
	{
		return m_pMapping->ModuleOk != 0;
	}

	uint32_t CIOModule_X20SI8110::getSerialNumber ()
	{
		return m_pMapping->SerialNumber;
	}

	uint16_t CIOModule_X20SI8110::getModuleID ()
	{
		return m_pMapping->ModuleID;
	}

	uint16_t CIOModule_X20SI8110::getHardwareVariant ()
	{
		return m_pMapping->HardwareVariant;
	}

	uint16_t CIOModule_X20SI8110::getFirmwareVersion ()
	{
		return m_pMapping->FirmwareVersion;
	}

	uint16_t CIOModule_X20SI8110::getInput (uint32_t nChannelNo)
	{
		switch (nChannelNo)
		{
			case 1:
				return m_pMapping->SafeDigitalInput01;
				break;

			case 2:
				return m_pMapping->SafeDigitalInput02;
				break;

			case 3:
				return m_pMapping->SafeDigitalInput03;
				break;

			case 4:
				return m_pMapping->SafeDigitalInput04;
				break;

			case 5:
				return m_pMapping->SafeDigitalInput05;
				break;

			case 6:
				return m_pMapping->SafeDigitalInput06;
				break;

			case 7:
				return m_pMapping->SafeDigitalInput07;
				break;

			case 8:
				return m_pMapping->SafeDigitalInput08;
				break;
			default:
				return 0;
				break;

		}
	}

	uint16_t CIOModule_X20SI8110::getDualInput (uint32_t nDualChannelNo)
	{

		switch (nDualChannelNo)
		{
			case 1:
				return m_pMapping->SafeTwoChannelInput0102;
				break;

			case 2:
				return m_pMapping->SafeTwoChannelInput0304;
				break;

			case 3:
				return m_pMapping->SafeTwoChannelInput0506;
				break;

			case 4:
				return m_pMapping->SafeTwoChannelInput0708;
				break;

			default:
				return 0;
				break;

		}

	}
	uint16_t CIOModule_X20SI8110::getSafeInputStatus (uint32_t nChannelNo)
	{
		switch (nChannelNo)
		{
			case 1:
				return m_pMapping->SafeInputOK01;
				break;

			case 2:
				return m_pMapping->SafeInputOK02;
				break;

			case 3:
				return m_pMapping->SafeInputOK03;
				break;

			case 4:
				return m_pMapping->SafeInputOK04;
				break;

			case 5:
				return m_pMapping->SafeInputOK05;
				break;

			case 6:
				return m_pMapping->SafeInputOK06;
				break;

			case 7:
				return m_pMapping->SafeInputOK07;
				break;

			case 8:
				return m_pMapping->SafeInputOK08;
				break;
			default:
				return 0;
				break;

		}
	}

	uint16_t CIOModule_X20SI8110::getSafeDualInputStatus (uint32_t nDualChannelNo)
	{
		switch (nDualChannelNo)
		{
			case 1:
				return m_pMapping->SafeTwoChannelOK0102;
				break;

			case 2:
				return m_pMapping->SafeTwoChannelOK0304;
				break;

			case 3:
				return m_pMapping->SafeTwoChannelOK0506;
				break;

			case 4:
				return m_pMapping->SafeTwoChannelOK0708;
				break;

			default:
				return 0;
				break;

		}
	}

}
```

#### IOModule_X20SI8110.hpp
```cpp
/*++

Copyright (C) 2024 Institute for Machine Tools and Industrial Management
TUM School of Engineering and Design
Technical University of Munich

All rights reserved.

Redistribution and use in source and binary forms, with or without
modification, are permitted provided that the following conditions are met:
	* Redistributions of source code must retain the above copyright
	  notice, this list of conditions and the following disclaimer.
	* Redistributions in binary form must reproduce the above copyright
	  notice, this list of conditions and the following disclaimer in the
	  documentation and/or other materials provided with the distribution.
	* Neither the name of the Technical University of Munich nor the
	  names of its contributors may be used to endorse or promote products
	  derived from this software without specific prior written permission.

THIS SOFTWARE IS PROVIDED BY THE COPYRIGHT HOLDERS AND CONTRIBUTORS "AS IS" AND
ANY EXPRESS OR IMPLIED WARRANTIES, INCLUDING, BUT NOT LIMITED TO, THE IMPLIED
WARRANTIES OF MERCHANTABILITY AND FITNESS FOR A PARTICULAR PURPOSE ARE
DISCLAIMED. IN NO EVENT SHALL TECHNICAL UNIVERSITY OF MUNICH BE LIABLE FOR ANY
DIRECT, INDIRECT, INCIDENTAL, SPECIAL, EXEMPLARY, OR CONSEQUENTIAL DAMAGES
(INCLUDING, BUT NOT LIMITED TO, PROCUREMENT OF SUBSTITUTE GOODS OR SERVICES;
LOSS OF USE, DATA, OR PROFITS; OR BUSINESS INTERRUPTION) HOWEVER CAUSED AND
ON ANY THEORY OF LIABILITY, WHETHER IN CONTRACT, STRICT LIABILITY, OR TORT
(INCLUDING NEGLIGENCE OR OTHERWISE) ARISING IN ANY WAY OUT OF THE USE OF THIS
SOFTWARE, EVEN IF ADVISED OF THE POSSIBILITY OF SUCH DAMAGE.

*/

#ifndef __IOMODULE_X20SI8110_HPP
#define __IOMODULE_X20SI8110_HPP

#include "../Framework/Framework.hpp"

namespace BuRCPP {

	class CIOModule_X20SI8110 : public CIOModule {
		protected:
		IOMappingX20SI8110_TYP * m_pMapping;

		public:
		CIOModule_X20SI8110 (const std::string & sName, IOMappingX20SI8110_TYP * pMapping);
		virtual ~CIOModule_X20SI8110 ();

		bool isActive () override;
		uint32_t getSerialNumber () override;
		uint16_t getModuleID () override;
		uint16_t getHardwareVariant () override;
		uint16_t getFirmwareVersion () override;

		uint16_t getInput (uint32_t);
		uint16_t getDualInput (uint32_t);
		uint16_t getSafeInputStatus (uint32_t);
		uint16_t getSafeDualInputStatus (uint32_t);

		void onRegisterJournal ();
		void onUpdateJournal ();

	};

}

#endif // __IOMODULE_X20SI8110_HPP
```

#### IOModule_X20SO6300.cpp
```cpp
/*++

Copyright (C) 2024 Institute for Machine Tools and Industrial Management
TUM School of Engineering and Design
Technical University of Munich

All rights reserved.

Redistribution and use in source and binary forms, with or without
modification, are permitted provided that the following conditions are met:
	* Redistributions of source code must retain the above copyright
	  notice, this list of conditions and the following disclaimer.
	* Redistributions in binary form must reproduce the above copyright
	  notice, this list of conditions and the following disclaimer in the
	  documentation and/or other materials provided with the distribution.
	* Neither the name of the Technical University of Munich nor the
	  names of its contributors may be used to endorse or promote products
	  derived from this software without specific prior written permission.

THIS SOFTWARE IS PROVIDED BY THE COPYRIGHT HOLDERS AND CONTRIBUTORS "AS IS" AND
ANY EXPRESS OR IMPLIED WARRANTIES, INCLUDING, BUT NOT LIMITED TO, THE IMPLIED
WARRANTIES OF MERCHANTABILITY AND FITNESS FOR A PARTICULAR PURPOSE ARE
DISCLAIMED. IN NO EVENT SHALL TECHNICAL UNIVERSITY OF MUNICH BE LIABLE FOR ANY
DIRECT, INDIRECT, INCIDENTAL, SPECIAL, EXEMPLARY, OR CONSEQUENTIAL DAMAGES
(INCLUDING, BUT NOT LIMITED TO, PROCUREMENT OF SUBSTITUTE GOODS OR SERVICES;
LOSS OF USE, DATA, OR PROFITS; OR BUSINESS INTERRUPTION) HOWEVER CAUSED AND
ON ANY THEORY OF LIABILITY, WHETHER IN CONTRACT, STRICT LIABILITY, OR TORT
(INCLUDING NEGLIGENCE OR OTHERWISE) ARISING IN ANY WAY OUT OF THE USE OF THIS
SOFTWARE, EVEN IF ADVISED OF THE POSSIBILITY OF SUCH DAMAGE.

*/

#include "IOModule_X20SO6300.hpp"

// Raw Registers
#define JOURNALVARIABLE_X20SO6300_MODULEOK 1
#define JOURNALVARIABLE_X20SO6300_SERIALNUMBER 2
#define JOURNALVARIABLE_X20SO6300_MODULEID 3
#define JOURNALVARIABLE_X20SO6300_HARDWAREVARIANT 4
#define JOURNALVARIABLE_X20SO6300_FIRMWAREVERSION 5
#define JOURNALVARIABLE_X20SO6300_SAFEMODULEOK 6
#define JOURNALVARIABLE_X20SO6300_SAFEDIGITALOUTPUT01 7
#define JOURNALVARIABLE_X20SO6300_SAFEDIGITALOUTPUT02 8
#define JOURNALVARIABLE_X20SO6300_SAFEDIGITALOUTPUT03 9
#define JOURNALVARIABLE_X20SO6300_SAFEDIGITALOUTPUT04 10
#define JOURNALVARIABLE_X20SO6300_SAFEDIGITALOUTPUT05 11
#define JOURNALVARIABLE_X20SO6300_SAFEDIGITALOUTPUT06 12
#define JOURNALVARIABLE_X20SO6300_SAFEOUTPUTOK01 13
#define JOURNALVARIABLE_X20SO6300_SAFEOUTPUTOK02 14
#define JOURNALVARIABLE_X20SO6300_SAFEOUTPUTOK03 15
#define JOURNALVARIABLE_X20SO6300_SAFEOUTPUTOK04 16
#define JOURNALVARIABLE_X20SO6300_SAFEOUTPUTOK05 17
#define JOURNALVARIABLE_X20SO6300_SAFEOUTPUTOK06 18

namespace BuRCPP {

	CIOModule_X20SO6300::CIOModule_X20SO6300 (const std::string & sName, IOMappingX20SO6300_TYP * pMapping)
		: CIOModule (sName), m_pMapping (pMapping)
	{

	}

	CIOModule_X20SO6300::~CIOModule_X20SO6300 ()
	{
	}

	void CIOModule_X20SO6300::onRegisterJournal ()
	{
		registerBoolValue ("ModuleOk", JOURNALVARIABLE_X20SO6300_MODULEOK);
		registerUInt32Value ("SerialNumber", JOURNALVARIABLE_X20SO6300_SERIALNUMBER);
		registerUInt16Value ("ModuleID", JOURNALVARIABLE_X20SO6300_MODULEID);
		registerUInt16Value ("HardwareVariant", JOURNALVARIABLE_X20SO6300_HARDWAREVARIANT);
		registerUInt16Value ("FirmwareVersion", JOURNALVARIABLE_X20SO6300_FIRMWAREVERSION);
		registerBoolValue ("SafeModuleOK", JOURNALVARIABLE_X20SO6300_SAFEMODULEOK);
		registerBoolValue ("SafeDigitalOutput01", JOURNALVARIABLE_X20SO6300_SAFEDIGITALOUTPUT01);
		registerBoolValue ("SafeDigitalOutput02", JOURNALVARIABLE_X20SO6300_SAFEDIGITALOUTPUT02);
		registerBoolValue ("SafeDigitalOutput03", JOURNALVARIABLE_X20SO6300_SAFEDIGITALOUTPUT03);
		registerBoolValue ("SafeDigitalOutput04", JOURNALVARIABLE_X20SO6300_SAFEDIGITALOUTPUT04);
		registerBoolValue ("SafeDigitalOutput05", JOURNALVARIABLE_X20SO6300_SAFEDIGITALOUTPUT05);
		registerBoolValue ("SafeDigitalOutput06", JOURNALVARIABLE_X20SO6300_SAFEDIGITALOUTPUT06);
		registerBoolValue ("SafeOutputOK01", JOURNALVARIABLE_X20SO6300_SAFEOUTPUTOK01);
		registerBoolValue ("SafeOutputOK02", JOURNALVARIABLE_X20SO6300_SAFEOUTPUTOK02);
		registerBoolValue ("SafeOutputOK03", JOURNALVARIABLE_X20SO6300_SAFEOUTPUTOK03);
		registerBoolValue ("SafeOutputOK04", JOURNALVARIABLE_X20SO6300_SAFEOUTPUTOK04);
		registerBoolValue ("SafeOutputOK05", JOURNALVARIABLE_X20SO6300_SAFEOUTPUTOK05);
		registerBoolValue ("SafeOutputOK06", JOURNALVARIABLE_X20SO6300_SAFEOUTPUTOK06);
	}

	void CIOModule_X20SO6300::onUpdateJournal ()
	{
		setBoolValue (JOURNALVARIABLE_X20SO6300_MODULEOK, m_pMapping->ModuleOk);
		setIntegerValue (JOURNALVARIABLE_X20SO6300_SERIALNUMBER, m_pMapping->SerialNumber);
		setIntegerValue (JOURNALVARIABLE_X20SO6300_MODULEID, m_pMapping->ModuleID);
		setIntegerValue (JOURNALVARIABLE_X20SO6300_HARDWAREVARIANT, m_pMapping->HardwareVariant);
		setIntegerValue (JOURNALVARIABLE_X20SO6300_FIRMWAREVERSION, m_pMapping->FirmwareVersion);
		setBoolValue (JOURNALVARIABLE_X20SO6300_SAFEMODULEOK, m_pMapping->SafeModuleOK);
		setBoolValue (JOURNALVARIABLE_X20SO6300_SAFEDIGITALOUTPUT01, m_pMapping->PhysicalStateOutput01);
		setBoolValue (JOURNALVARIABLE_X20SO6300_SAFEDIGITALOUTPUT02, m_pMapping->PhysicalStateOutput02);
		setBoolValue (JOURNALVARIABLE_X20SO6300_SAFEDIGITALOUTPUT03, m_pMapping->PhysicalStateOutput03);
		setBoolValue (JOURNALVARIABLE_X20SO6300_SAFEDIGITALOUTPUT04, m_pMapping->PhysicalStateOutput04);
		setBoolValue (JOURNALVARIABLE_X20SO6300_SAFEDIGITALOUTPUT05, m_pMapping->PhysicalStateOutput05);
		setBoolValue (JOURNALVARIABLE_X20SO6300_SAFEDIGITALOUTPUT06, m_pMapping->PhysicalStateOutput06);
		setBoolValue (JOURNALVARIABLE_X20SO6300_SAFEOUTPUTOK01, m_pMapping->SafeOutputOK01);
		setBoolValue (JOURNALVARIABLE_X20SO6300_SAFEOUTPUTOK02, m_pMapping->SafeOutputOK02);
		setBoolValue (JOURNALVARIABLE_X20SO6300_SAFEOUTPUTOK03, m_pMapping->SafeOutputOK03);
		setBoolValue (JOURNALVARIABLE_X20SO6300_SAFEOUTPUTOK04, m_pMapping->SafeOutputOK04);
		setBoolValue (JOURNALVARIABLE_X20SO6300_SAFEOUTPUTOK05, m_pMapping->SafeOutputOK05);
		setBoolValue (JOURNALVARIABLE_X20SO6300_SAFEOUTPUTOK06, m_pMapping->SafeOutputOK06);
	}

	bool CIOModule_X20SO6300::isActive ()
	{
		return m_pMapping->ModuleOk != 0;
	}

	uint32_t CIOModule_X20SO6300::getSerialNumber ()
	{
		return m_pMapping->SerialNumber;
	}

	uint16_t CIOModule_X20SO6300::getModuleID ()
	{
		return m_pMapping->ModuleID;
	}

	uint16_t CIOModule_X20SO6300::getHardwareVariant ()
	{
		return m_pMapping->HardwareVariant;
	}

	uint16_t CIOModule_X20SO6300::getFirmwareVersion ()
	{
		return m_pMapping->FirmwareVersion;
	}

	uint16_t CIOModule_X20SO6300::getPhysicalStateOutput (uint32_t nChannelNo)
	{
		switch (nChannelNo)
		{
			case 1:
				return m_pMapping->PhysicalStateOutput01;
				break;

			case 2:
				return m_pMapping->PhysicalStateOutput02;
				break;

			case 3:
				return m_pMapping->PhysicalStateOutput03;
				break;

			case 4:
				return m_pMapping->PhysicalStateOutput04;
				break;

			case 5:
				return m_pMapping->PhysicalStateOutput05;
				break;

			case 6:
				return m_pMapping->PhysicalStateOutput06;
				break;
			default:
				return 0;
				break;

		}
	}

	uint16_t CIOModule_X20SO6300::getSafeOutputStatus (uint32_t nChannelNo)
	{
		switch (nChannelNo)
		{
			case 1:
				return m_pMapping->SafeOutputOK01;
				break;

			case 2:
				return m_pMapping->SafeOutputOK02;
				break;

			case 3:
				return m_pMapping->SafeOutputOK03;
				break;

			case 4:
				return m_pMapping->SafeOutputOK04;
				break;

			case 5:
				return m_pMapping->SafeOutputOK05;
				break;

			case 6:
				return m_pMapping->SafeOutputOK06;
				break;
			default:
				return 0;
				break;

		}
	}

}
```

#### IOModule_X20SO6300.hpp
```cpp
/*++

Copyright (C) 2024 Institute for Machine Tools and Industrial Management
TUM School of Engineering and Design
Technical University of Munich

All rights reserved.

Redistribution and use in source and binary forms, with or without
modification, are permitted provided that the following conditions are met:
	* Redistributions of source code must retain the above copyright
	  notice, this list of conditions and the following disclaimer.
	* Redistributions in binary form must reproduce the above copyright
	  notice, this list of conditions and the following disclaimer in the
	  documentation and/or other materials provided with the distribution.
	* Neither the name of the Technical University of Munich nor the
	  names of its contributors may be used to endorse or promote products
	  derived from this software without specific prior written permission.

THIS SOFTWARE IS PROVIDED BY THE COPYRIGHT HOLDERS AND CONTRIBUTORS "AS IS" AND
ANY EXPRESS OR IMPLIED WARRANTIES, INCLUDING, BUT NOT LIMITED TO, THE IMPLIED
WARRANTIES OF MERCHANTABILITY AND FITNESS FOR A PARTICULAR PURPOSE ARE
DISCLAIMED. IN NO EVENT SHALL TECHNICAL UNIVERSITY OF MUNICH BE LIABLE FOR ANY
DIRECT, INDIRECT, INCIDENTAL, SPECIAL, EXEMPLARY, OR CONSEQUENTIAL DAMAGES
(INCLUDING, BUT NOT LIMITED TO, PROCUREMENT OF SUBSTITUTE GOODS OR SERVICES;
LOSS OF USE, DATA, OR PROFITS; OR BUSINESS INTERRUPTION) HOWEVER CAUSED AND
ON ANY THEORY OF LIABILITY, WHETHER IN CONTRACT, STRICT LIABILITY, OR TORT
(INCLUDING NEGLIGENCE OR OTHERWISE) ARISING IN ANY WAY OUT OF THE USE OF THIS
SOFTWARE, EVEN IF ADVISED OF THE POSSIBILITY OF SUCH DAMAGE.

*/

#ifndef __IOMODULE_X20SO6300_HPP
#define __IOMODULE_X20SO6300_HPP

#include "../Framework/Framework.hpp"

namespace BuRCPP {

	class CIOModule_X20SO6300 : public CIOModule {
		protected:
		IOMappingX20SO6300_TYP * m_pMapping;

		public:
		CIOModule_X20SO6300 (const std::string & sName, IOMappingX20SO6300_TYP * pMapping);
		virtual ~CIOModule_X20SO6300 ();

		bool isActive () override;
		uint32_t getSerialNumber () override;
		uint16_t getModuleID () override;
		uint16_t getHardwareVariant () override;
		uint16_t getFirmwareVersion () override;

		uint16_t getPhysicalStateOutput (uint32_t);
		uint16_t getSafeOutputStatus (uint32_t);

		void onRegisterJournal ();
		void onUpdateJournal ();

	};

}

#endif // __IOMODULE_X20SO6300_HPP
```

#### IOModule_X20SC0842.cpp
```cpp
/*++

Copyright (C) 2024 Institute for Machine Tools and Industrial Management
TUM School of Engineering and Design
Technical University of Munich

All rights reserved.

Redistribution and use in source and binary forms, with or without
modification, are permitted provided that the following conditions are met:
	* Redistributions of source code must retain the above copyright
	  notice, this list of conditions and the following disclaimer.
	* Redistributions in binary form must reproduce the above copyright
	  notice, this list of conditions and the following disclaimer in the
	  documentation and/or other materials provided with the distribution.
	* Neither the name of the Technical University of Munich nor the
	  names of its contributors may be used to endorse or promote products
	  derived from this software without specific prior written permission.

THIS SOFTWARE IS PROVIDED BY THE COPYRIGHT HOLDERS AND CONTRIBUTORS "AS IS" AND
ANY EXPRESS OR IMPLIED WARRANTIES, INCLUDING, BUT NOT LIMITED TO, THE IMPLIED
WARRANTIES OF MERCHANTABILITY AND FITNESS FOR A PARTICULAR PURPOSE ARE
DISCLAIMED. IN NO EVENT SHALL TECHNICAL UNIVERSITY OF MUNICH BE LIABLE FOR ANY
DIRECT, INDIRECT, INCIDENTAL, SPECIAL, EXEMPLARY, OR CONSEQUENTIAL DAMAGES
(INCLUDING, BUT NOT LIMITED TO, PROCUREMENT OF SUBSTITUTE GOODS OR SERVICES;
LOSS OF USE, DATA, OR PROFITS; OR BUSINESS INTERRUPTION) HOWEVER CAUSED AND
ON ANY THEORY OF LIABILITY, WHETHER IN CONTRACT, STRICT LIABILITY, OR TORT
(INCLUDING NEGLIGENCE OR OTHERWISE) ARISING IN ANY WAY OUT OF THE USE OF THIS
SOFTWARE, EVEN IF ADVISED OF THE POSSIBILITY OF SUCH DAMAGE.

*/
#include "IOModule_X20SC0842.hpp"

// Raw Registers
#define JOURNALVARIABLE_X20SC0842_MODULEOK 1
#define JOURNALVARIABLE_X20SC0842_SERIALNUMBER 2
#define JOURNALVARIABLE_X20SC0842_MODULEID 3
#define JOURNALVARIABLE_X20SC0842_HARDWAREVARIANT 4
#define JOURNALVARIABLE_X20SC0842_FIRMWAREVERSION 5
#define JOURNALVARIABLE_X20SC0842_SAFEMODULEOK 6
#define JOURNALVARIABLE_X20SC0842_SAFEDIGITALOUTPUT01 7
#define JOURNALVARIABLE_X20SC0842_SAFEDIGITALOUTPUT02 8
#define JOURNALVARIABLE_X20SC0842_SAFEDIGITALOUTPUT03 9
#define JOURNALVARIABLE_X20SC0842_SAFEDIGITALOUTPUT04 10
#define JOURNALVARIABLE_X20SC0842_SAFEDIGITALOUTPUT05 11
#define JOURNALVARIABLE_X20SC0842_SAFEDIGITALOUTPUT06 12
#define JOURNALVARIABLE_X20SC0842_SAFEOUTPUTOK01 13
#define JOURNALVARIABLE_X20SC0842_SAFEOUTPUTOK02 14
#define JOURNALVARIABLE_X20SC0842_SAFEOUTPUTOK03 15
#define JOURNALVARIABLE_X20SC0842_SAFEOUTPUTOK04 16
#define JOURNALVARIABLE_X20SC0842_SAFEOUTPUTOK05 17
#define JOURNALVARIABLE_X20SC0842_SAFEOUTPUTOK06 18
#define JOURNALVARIABLE_X20SC0842_SAFEDIGITALINPUT01 19
#define JOURNALVARIABLE_X20SC0842_SAFEDIGITALINPUT02 20
#define JOURNALVARIABLE_X20SC0842_SAFEDIGITALINPUT03 21
#define JOURNALVARIABLE_X20SC0842_SAFEDIGITALINPUT04 22
#define JOURNALVARIABLE_X20SC0842_SAFEDIGITALINPUT05 23
#define JOURNALVARIABLE_X20SC0842_SAFEDIGITALINPUT06 24
#define JOURNALVARIABLE_X20SC0842_SAFEDIGITALINPUT07 25
#define JOURNALVARIABLE_X20SC0842_SAFEDIGITALINPUT08 26
#define JOURNALVARIABLE_X20SC0842_SAFETWOCHANNELINPUT0102 27
#define JOURNALVARIABLE_X20SC0842_SAFETWOCHANNELINPUT0304 28
#define JOURNALVARIABLE_X20SC0842_SAFETWOCHANNELINPUT0506 29
#define JOURNALVARIABLE_X20SC0842_SAFETWOCHANNELINPUT0708 30
#define JOURNALVARIABLE_X20SC0842_SAFEINPUTOK01 31
#define JOURNALVARIABLE_X20SC0842_SAFEINPUTOK02 32
#define JOURNALVARIABLE_X20SC0842_SAFEINPUTOK03 33
#define JOURNALVARIABLE_X20SC0842_SAFEINPUTOK04 34
#define JOURNALVARIABLE_X20SC0842_SAFEINPUTOK05 35
#define JOURNALVARIABLE_X20SC0842_SAFEINPUTOK06 36
#define JOURNALVARIABLE_X20SC0842_SAFEINPUTOK07 37
#define JOURNALVARIABLE_X20SC0842_SAFEINPUTOK08 38
#define JOURNALVARIABLE_X20SC0842_SAFETWOCHANNELOK0102 39
#define JOURNALVARIABLE_X20SC0842_SAFETWOCHANNELOK0304 40
#define JOURNALVARIABLE_X20SC0842_SAFETWOCHANNELOK0506 41
#define JOURNALVARIABLE_X20SC0842_SAFETWOCHANNELOK0708 42

namespace BuRCPP {

	CIOModule_X20SC0842::CIOModule_X20SC0842 (const std::string & sName, IOMappingX20SC0842_TYP * pMapping)
		: CIOModule (sName), m_pMapping (pMapping)
	{

	}

	CIOModule_X20SC0842::~CIOModule_X20SC0842 ()
	{
	}

	void CIOModule_X20SC0842::onRegisterJournal ()
	{
		registerBoolValue ("ModuleOk", JOURNALVARIABLE_X20SC0842_MODULEOK);
		registerUInt32Value ("SerialNumber", JOURNALVARIABLE_X20SC0842_SERIALNUMBER);
		registerUInt16Value ("ModuleID", JOURNALVARIABLE_X20SC0842_MODULEID);
		registerUInt16Value ("HardwareVariant", JOURNALVARIABLE_X20SC0842_HARDWAREVARIANT);
		registerUInt16Value ("FirmwareVersion", JOURNALVARIABLE_X20SC0842_FIRMWAREVERSION);
		registerBoolValue ("SafeModuleOK", JOURNALVARIABLE_X20SC0842_SAFEMODULEOK);
		registerBoolValue ("SafeDigitalOutput01", JOURNALVARIABLE_X20SC0842_SAFEDIGITALOUTPUT01);
		registerBoolValue ("SafeDigitalOutput02", JOURNALVARIABLE_X20SC0842_SAFEDIGITALOUTPUT02);
		registerBoolValue ("SafeDigitalOutput03", JOURNALVARIABLE_X20SC0842_SAFEDIGITALOUTPUT03);
		registerBoolValue ("SafeDigitalOutput04", JOURNALVARIABLE_X20SC0842_SAFEDIGITALOUTPUT04);
		registerBoolValue ("SafeDigitalOutput05", JOURNALVARIABLE_X20SC0842_SAFEDIGITALOUTPUT05);
		registerBoolValue ("SafeDigitalOutput06", JOURNALVARIABLE_X20SC0842_SAFEDIGITALOUTPUT06);
		registerBoolValue ("SafeOutputOK01", JOURNALVARIABLE_X20SC0842_SAFEOUTPUTOK01);
		registerBoolValue ("SafeOutputOK02", JOURNALVARIABLE_X20SC0842_SAFEOUTPUTOK02);
		registerBoolValue ("SafeOutputOK03", JOURNALVARIABLE_X20SC0842_SAFEOUTPUTOK03);
		registerBoolValue ("SafeOutputOK04", JOURNALVARIABLE_X20SC0842_SAFEOUTPUTOK04);
		registerBoolValue ("SafeOutputOK05", JOURNALVARIABLE_X20SC0842_SAFEOUTPUTOK05);
		registerBoolValue ("SafeOutputOK06", JOURNALVARIABLE_X20SC0842_SAFEOUTPUTOK06);
		registerBoolValue ("SafeDigitalInput01", JOURNALVARIABLE_X20SC0842_SAFEDIGITALINPUT01);
		registerBoolValue ("SafeDigitalInput02", JOURNALVARIABLE_X20SC0842_SAFEDIGITALINPUT02);
		registerBoolValue ("SafeDigitalInput03", JOURNALVARIABLE_X20SC0842_SAFEDIGITALINPUT03);
		registerBoolValue ("SafeDigitalInput04", JOURNALVARIABLE_X20SC0842_SAFEDIGITALINPUT04);
		registerBoolValue ("SafeDigitalInput05", JOURNALVARIABLE_X20SC0842_SAFEDIGITALINPUT05);
		registerBoolValue ("SafeDigitalInput06", JOURNALVARIABLE_X20SC0842_SAFEDIGITALINPUT06);
		registerBoolValue ("SafeDigitalInput07", JOURNALVARIABLE_X20SC0842_SAFEDIGITALINPUT07);
		registerBoolValue ("SafeDigitalInput08", JOURNALVARIABLE_X20SC0842_SAFEDIGITALINPUT08);
		registerBoolValue ("SafeTwoChannelInput0102", JOURNALVARIABLE_X20SC0842_SAFETWOCHANNELINPUT0102);
		registerBoolValue ("SafeTwoChannelInput0304", JOURNALVARIABLE_X20SC0842_SAFETWOCHANNELINPUT0304);
		registerBoolValue ("SafeTwoChannelInput0506", JOURNALVARIABLE_X20SC0842_SAFETWOCHANNELINPUT0506);
		registerBoolValue ("SafeTwoChannelInput0708", JOURNALVARIABLE_X20SC0842_SAFETWOCHANNELINPUT0708);
		registerBoolValue ("SafeInputOK01", JOURNALVARIABLE_X20SC0842_SAFEINPUTOK01);
		registerBoolValue ("SafeInputOK02", JOURNALVARIABLE_X20SC0842_SAFEINPUTOK02);
		registerBoolValue ("SafeInputOK03", JOURNALVARIABLE_X20SC0842_SAFEINPUTOK03);
		registerBoolValue ("SafeInputOK04", JOURNALVARIABLE_X20SC0842_SAFEINPUTOK04);
		registerBoolValue ("SafeInputOK05", JOURNALVARIABLE_X20SC0842_SAFEINPUTOK05);
		registerBoolValue ("SafeInputOK06", JOURNALVARIABLE_X20SC0842_SAFEINPUTOK06);
		registerBoolValue ("SafeInputOK07", JOURNALVARIABLE_X20SC0842_SAFEINPUTOK07);
		registerBoolValue ("SafeInputOK08", JOURNALVARIABLE_X20SC0842_SAFEINPUTOK08);
		registerBoolValue ("SafeTwoChannelOK0102", JOURNALVARIABLE_X20SC0842_SAFETWOCHANNELOK0102);
		registerBoolValue ("SafeTwoChannelOK0304", JOURNALVARIABLE_X20SC0842_SAFETWOCHANNELOK0304);
		registerBoolValue ("SafeTwoChannelOK0506", JOURNALVARIABLE_X20SC0842_SAFETWOCHANNELOK0506);
		registerBoolValue ("SafeTwoChannelOK0708", JOURNALVARIABLE_X20SC0842_SAFETWOCHANNELOK0708);
	}

	void CIOModule_X20SC0842::onUpdateJournal ()
	{
		setBoolValue (JOURNALVARIABLE_X20SC0842_MODULEOK, m_pMapping->ModuleOk);
		setIntegerValue (JOURNALVARIABLE_X20SC0842_SERIALNUMBER, m_pMapping->SerialNumber);
		setIntegerValue (JOURNALVARIABLE_X20SC0842_MODULEID, m_pMapping->ModuleID);
		setIntegerValue (JOURNALVARIABLE_X20SC0842_HARDWAREVARIANT, m_pMapping->HardwareVariant);
		setIntegerValue (JOURNALVARIABLE_X20SC0842_FIRMWAREVERSION, m_pMapping->FirmwareVersion);
		setBoolValue (JOURNALVARIABLE_X20SC0842_SAFEMODULEOK, m_pMapping->SafeModuleOK);
		setBoolValue (JOURNALVARIABLE_X20SC0842_SAFEDIGITALOUTPUT01, m_pMapping->PhysicalStateOutput01);
		setBoolValue (JOURNALVARIABLE_X20SC0842_SAFEDIGITALOUTPUT02, m_pMapping->PhysicalStateOutput02);
		setBoolValue (JOURNALVARIABLE_X20SC0842_SAFEDIGITALOUTPUT03, m_pMapping->PhysicalStateOutput03);
		setBoolValue (JOURNALVARIABLE_X20SC0842_SAFEDIGITALOUTPUT04, m_pMapping->PhysicalStateOutput04);
		setBoolValue (JOURNALVARIABLE_X20SC0842_SAFEDIGITALOUTPUT05, m_pMapping->PhysicalStateOutput05);
		setBoolValue (JOURNALVARIABLE_X20SC0842_SAFEDIGITALOUTPUT06, m_pMapping->PhysicalStateOutput06);
		setBoolValue (JOURNALVARIABLE_X20SC0842_SAFEOUTPUTOK01, m_pMapping->SafeOutputOK01);
		setBoolValue (JOURNALVARIABLE_X20SC0842_SAFEOUTPUTOK02, m_pMapping->SafeOutputOK02);
		setBoolValue (JOURNALVARIABLE_X20SC0842_SAFEOUTPUTOK03, m_pMapping->SafeOutputOK03);
		setBoolValue (JOURNALVARIABLE_X20SC0842_SAFEOUTPUTOK04, m_pMapping->SafeOutputOK04);
		setBoolValue (JOURNALVARIABLE_X20SC0842_SAFEOUTPUTOK05, m_pMapping->SafeOutputOK05);
		setBoolValue (JOURNALVARIABLE_X20SC0842_SAFEOUTPUTOK06, m_pMapping->SafeOutputOK06);
		setBoolValue (JOURNALVARIABLE_X20SC0842_SAFEDIGITALINPUT01, m_pMapping->SafeDigitalInput01);
		setBoolValue (JOURNALVARIABLE_X20SC0842_SAFEDIGITALINPUT02, m_pMapping->SafeDigitalInput02);
		setBoolValue (JOURNALVARIABLE_X20SC0842_SAFEDIGITALINPUT03, m_pMapping->SafeDigitalInput03);
		setBoolValue (JOURNALVARIABLE_X20SC0842_SAFEDIGITALINPUT04, m_pMapping->SafeDigitalInput04);
		setBoolValue (JOURNALVARIABLE_X20SC0842_SAFEDIGITALINPUT05, m_pMapping->SafeDigitalInput05);
		setBoolValue (JOURNALVARIABLE_X20SC0842_SAFEDIGITALINPUT06, m_pMapping->SafeDigitalInput06);
		setBoolValue (JOURNALVARIABLE_X20SC0842_SAFEDIGITALINPUT07, m_pMapping->SafeDigitalInput07);
		setBoolValue (JOURNALVARIABLE_X20SC0842_SAFEDIGITALINPUT08, m_pMapping->SafeDigitalInput08);
		setBoolValue (JOURNALVARIABLE_X20SC0842_SAFETWOCHANNELINPUT0102, m_pMapping->SafeTwoChannelInput0102);
		setBoolValue (JOURNALVARIABLE_X20SC0842_SAFETWOCHANNELINPUT0304, m_pMapping->SafeTwoChannelInput0304);
		setBoolValue (JOURNALVARIABLE_X20SC0842_SAFETWOCHANNELINPUT0506, m_pMapping->SafeTwoChannelInput0506);
		setBoolValue (JOURNALVARIABLE_X20SC0842_SAFETWOCHANNELINPUT0708, m_pMapping->SafeTwoChannelInput0708);
		setBoolValue (JOURNALVARIABLE_X20SC0842_SAFEINPUTOK01, m_pMapping->SafeInputOK01);
		setBoolValue (JOURNALVARIABLE_X20SC0842_SAFEINPUTOK02, m_pMapping->SafeInputOK02);
		setBoolValue (JOURNALVARIABLE_X20SC0842_SAFEINPUTOK03, m_pMapping->SafeInputOK03);
		setBoolValue (JOURNALVARIABLE_X20SC0842_SAFEINPUTOK04, m_pMapping->SafeInputOK04);
		setBoolValue (JOURNALVARIABLE_X20SC0842_SAFEINPUTOK05, m_pMapping->SafeInputOK05);
		setBoolValue (JOURNALVARIABLE_X20SC0842_SAFEINPUTOK06, m_pMapping->SafeInputOK06);
		setBoolValue (JOURNALVARIABLE_X20SC0842_SAFEINPUTOK07, m_pMapping->SafeInputOK07);
		setBoolValue (JOURNALVARIABLE_X20SC0842_SAFEINPUTOK08, m_pMapping->SafeInputOK08);
		setBoolValue (JOURNALVARIABLE_X20SC0842_SAFETWOCHANNELOK0102, m_pMapping->SafeTwoChannelOK0102);
		setBoolValue (JOURNALVARIABLE_X20SC0842_SAFETWOCHANNELOK0304, m_pMapping->SafeTwoChannelOK0304);
		setBoolValue (JOURNALVARIABLE_X20SC0842_SAFETWOCHANNELOK0506, m_pMapping->SafeTwoChannelOK0506);
		setBoolValue (JOURNALVARIABLE_X20SC0842_SAFETWOCHANNELOK0708, m_pMapping->SafeTwoChannelOK0708);
	}

	bool CIOModule_X20SC0842::isActive ()
	{
		return m_pMapping->ModuleOk != 0;
	}

	uint32_t CIOModule_X20SC0842::getSerialNumber ()
	{
		return m_pMapping->SerialNumber;
	}

	uint16_t CIOModule_X20SC0842::getModuleID ()
	{
		return m_pMapping->ModuleID;
	}

	uint16_t CIOModule_X20SC0842::getHardwareVariant ()
	{
		return m_pMapping->HardwareVariant;
	}

	uint16_t CIOModule_X20SC0842::getFirmwareVersion ()
	{
		return m_pMapping->FirmwareVersion;
	}

	uint16_t CIOModule_X20SC0842::getPhysicalStateOutput (uint32_t nChannelNo)
	{
		switch (nChannelNo)
		{
			case 1:
				return m_pMapping->PhysicalStateOutput01;
				break;

			case 2:
				return m_pMapping->PhysicalStateOutput02;
				break;

			case 3:
				return m_pMapping->PhysicalStateOutput03;
				break;

			case 4:
				return m_pMapping->PhysicalStateOutput04;
				break;

			case 5:
				return m_pMapping->PhysicalStateOutput05;
				break;

			case 6:
				return m_pMapping->PhysicalStateOutput06;
				break;
			default:
				return 0;
				break;

		}
	}

	uint16_t CIOModule_X20SC0842::getSafeOutputStatus (uint32_t nChannelNo)
	{
		switch (nChannelNo)
		{
			case 1:
				return m_pMapping->SafeOutputOK01;
				break;

			case 2:
				return m_pMapping->SafeOutputOK02;
				break;

			case 3:
				return m_pMapping->SafeOutputOK03;
				break;

			case 4:
				return m_pMapping->SafeOutputOK04;
				break;

			case 5:
				return m_pMapping->SafeOutputOK05;
				break;

			case 6:
				return m_pMapping->SafeOutputOK06;
				break;
			default:
				return 0;
				break;

		}
	}

	uint16_t CIOModule_X20SC0842::getInput (uint32_t nChannelNo)
	{
		switch (nChannelNo)
		{
			case 1:
				return m_pMapping->SafeDigitalInput01;
				break;

			case 2:
				return m_pMapping->SafeDigitalInput02;
				break;

			case 3:
				return m_pMapping->SafeDigitalInput03;
				break;

			case 4:
				return m_pMapping->SafeDigitalInput04;
				break;

			case 5:
				return m_pMapping->SafeDigitalInput05;
				break;

			case 6:
				return m_pMapping->SafeDigitalInput06;
				break;

			case 7:
				return m_pMapping->SafeDigitalInput07;
				break;

			case 8:
				return m_pMapping->SafeDigitalInput08;
				break;
			default:
				return 0;
				break;

		}
	}

	uint16_t CIOModule_X20SC0842::getDualInput (uint32_t nDualChannelNo)
	{

		switch (nDualChannelNo)
		{
			case 1:
				return m_pMapping->SafeTwoChannelInput0102;
				break;

			case 2:
				return m_pMapping->SafeTwoChannelInput0304;
				break;

			case 3:
				return m_pMapping->SafeTwoChannelInput0506;
				break;

			case 4:
				return m_pMapping->SafeTwoChannelInput0708;
				break;

			default:
				return 0;
				break;

		}

	}
	uint16_t CIOModule_X20SC0842::getSafeInputStatus (uint32_t nChannelNo)
	{
		switch (nChannelNo)
		{
			case 1:
				return m_pMapping->SafeInputOK01;
				break;

			case 2:
				return m_pMapping->SafeInputOK02;
				break;

			case 3:
				return m_pMapping->SafeInputOK03;
				break;

			case 4:
				return m_pMapping->SafeInputOK04;
				break;

			case 5:
				return m_pMapping->SafeInputOK05;
				break;

			case 6:
				return m_pMapping->SafeInputOK06;
				break;

			case 7:
				return m_pMapping->SafeInputOK07;
				break;

			case 8:
				return m_pMapping->SafeInputOK08;
				break;
			default:
				return 0;
				break;

		}
	}

	uint16_t CIOModule_X20SC0842::getSafeDualInputStatus (uint32_t nDualChannelNo)
	{
		switch (nDualChannelNo)
		{
			case 1:
				return m_pMapping->SafeTwoChannelOK0102;
				break;

			case 2:
				return m_pMapping->SafeTwoChannelOK0304;
				break;

			case 3:
				return m_pMapping->SafeTwoChannelOK0506;
				break;

			case 4:
				return m_pMapping->SafeTwoChannelOK0708;
				break;

			default:
				return 0;
				break;

		}

	}
}
```

#### IOModule_X20SC0842.hpp
```cpp
/*++

Copyright (C) 2024 Institute for Machine Tools and Industrial Management
TUM School of Engineering and Design
Technical University of Munich

All rights reserved.

Redistribution and use in source and binary forms, with or without
modification, are permitted provided that the following conditions are met:
	* Redistributions of source code must retain the above copyright
	  notice, this list of conditions and the following disclaimer.
	* Redistributions in binary form must reproduce the above copyright
	  notice, this list of conditions and the following disclaimer in the
	  documentation and/or other materials provided with the distribution.
	* Neither the name of the Technical University of Munich nor the
	  names of its contributors may be used to endorse or promote products
	  derived from this software without specific prior written permission.

THIS SOFTWARE IS PROVIDED BY THE COPYRIGHT HOLDERS AND CONTRIBUTORS "AS IS" AND
ANY EXPRESS OR IMPLIED WARRANTIES, INCLUDING, BUT NOT LIMITED TO, THE IMPLIED
WARRANTIES OF MERCHANTABILITY AND FITNESS FOR A PARTICULAR PURPOSE ARE
DISCLAIMED. IN NO EVENT SHALL TECHNICAL UNIVERSITY OF MUNICH BE LIABLE FOR ANY
DIRECT, INDIRECT, INCIDENTAL, SPECIAL, EXEMPLARY, OR CONSEQUENTIAL DAMAGES
(INCLUDING, BUT NOT LIMITED TO, PROCUREMENT OF SUBSTITUTE GOODS OR SERVICES;
LOSS OF USE, DATA, OR PROFITS; OR BUSINESS INTERRUPTION) HOWEVER CAUSED AND
ON ANY THEORY OF LIABILITY, WHETHER IN CONTRACT, STRICT LIABILITY, OR TORT
(INCLUDING NEGLIGENCE OR OTHERWISE) ARISING IN ANY WAY OUT OF THE USE OF THIS
SOFTWARE, EVEN IF ADVISED OF THE POSSIBILITY OF SUCH DAMAGE.

*/

#ifndef __IOMODULE_X20SC0842_HPP
#define __IOMODULE_X20SC0842_HPP

#include "../Framework/Framework.hpp"

namespace BuRCPP {

	class CIOModule_X20SC0842 : public CIOModule {
		protected:
		IOMappingX20SC0842_TYP * m_pMapping;

		public:
		CIOModule_X20SC0842 (const std::string & sName, IOMappingX20SC0842_TYP * pMapping);
		virtual ~CIOModule_X20SC0842 ();

		bool isActive () override;
		uint32_t getSerialNumber () override;
		uint16_t getModuleID () override;
		uint16_t getHardwareVariant () override;
		uint16_t getFirmwareVersion () override;

		uint16_t getInput (uint32_t);
		uint16_t getDualInput (uint32_t);
		uint16_t getSafeInputStatus (uint32_t);
		uint16_t getPhysicalStateOutput (uint32_t);
		uint16_t getSafeDualInputStatus (uint32_t);
		uint16_t getSafeOutputStatus (uint32_t);

		void onRegisterJournal ();
		void onUpdateJournal ();

	};

}

#endif // __IOMODULE_X20SC0842_HPP
```

#### IOModule_X20DO6322.hpp
```cpp
/*++

Copyright (C) 2024 Institute for Machine Tools and Industrial Management
TUM School of Engineering and Design
Technical University of Munich

All rights reserved.

Redistribution and use in source and binary forms, with or without
modification, are permitted provided that the following conditions are met:
	* Redistributions of source code must retain the above copyright
	  notice, this list of conditions and the following disclaimer.
	* Redistributions in binary form must reproduce the above copyright
	  notice, this list of conditions and the following disclaimer in the
	  documentation and/or other materials provided with the distribution.
	* Neither the name of the Technical University of Munich nor the
	  names of its contributors may be used to endorse or promote products
	  derived from this software without specific prior written permission.

THIS SOFTWARE IS PROVIDED BY THE COPYRIGHT HOLDERS AND CONTRIBUTORS "AS IS" AND
ANY EXPRESS OR IMPLIED WARRANTIES, INCLUDING, BUT NOT LIMITED TO, THE IMPLIED
WARRANTIES OF MERCHANTABILITY AND FITNESS FOR A PARTICULAR PURPOSE ARE
DISCLAIMED. IN NO EVENT SHALL TECHNICAL UNIVERSITY OF MUNICH BE LIABLE FOR ANY
DIRECT, INDIRECT, INCIDENTAL, SPECIAL, EXEMPLARY, OR CONSEQUENTIAL DAMAGES
(INCLUDING, BUT NOT LIMITED TO, PROCUREMENT OF SUBSTITUTE GOODS OR SERVICES;
LOSS OF USE, DATA, OR PROFITS; OR BUSINESS INTERRUPTION) HOWEVER CAUSED AND
ON ANY THEORY OF LIABILITY, WHETHER IN CONTRACT, STRICT LIABILITY, OR TORT
(INCLUDING NEGLIGENCE OR OTHERWISE) ARISING IN ANY WAY OUT OF THE USE OF THIS
SOFTWARE, EVEN IF ADVISED OF THE POSSIBILITY OF SUCH DAMAGE.

*/
#ifndef __IOMODULE_X20DO6322_HPP
#define __IOMODULE_X20DO6322_HPP

#include "../Framework/Framework.hpp"

namespace BuRCPP {

	class CIOModule_X20DO6322 : public CIOModule {
		protected:
		IOMappingX20DO6322_TYP * m_pMapping;

		public:
		CIOModule_X20DO6322 (const std::string & sName, IOMappingX20DO6322_TYP * pMapping);
		virtual ~CIOModule_X20DO6322 ();

		bool isActive () override;
		uint32_t getSerialNumber () override;
		uint16_t getModuleID () override;
		uint16_t getHardwareVariant () override;
		uint16_t getFirmwareVersion () override;

		void setOutput (uint32_t, bool);

		uint16_t getIOStatus (uint32_t);

		void onRegisterJournal ();
		void onUpdateJournal ();
		bool getOutput (uint32_t nChannelNo);

	};

}

#endif // __IOMODULE_X20DO6322_HPP
```

#### IOModule_X20DO6322.cpp
```cpp
/*++

Copyright (C) 2024 Institute for Machine Tools and Industrial Management
TUM School of Engineering and Design
Technical University of Munich

All rights reserved.

Redistribution and use in source and binary forms, with or without
modification, are permitted provided that the following conditions are met:
	* Redistributions of source code must retain the above copyright
	  notice, this list of conditions and the following disclaimer.
	* Redistributions in binary form must reproduce the above copyright
	  notice, this list of conditions and the following disclaimer in the
	  documentation and/or other materials provided with the distribution.
	* Neither the name of the Technical University of Munich nor the
	  names of its contributors may be used to endorse or promote products
	  derived from this software without specific prior written permission.

THIS SOFTWARE IS PROVIDED BY THE COPYRIGHT HOLDERS AND CONTRIBUTORS "AS IS" AND
ANY EXPRESS OR IMPLIED WARRANTIES, INCLUDING, BUT NOT LIMITED TO, THE IMPLIED
WARRANTIES OF MERCHANTABILITY AND FITNESS FOR A PARTICULAR PURPOSE ARE
DISCLAIMED. IN NO EVENT SHALL TECHNICAL UNIVERSITY OF MUNICH BE LIABLE FOR ANY
DIRECT, INDIRECT, INCIDENTAL, SPECIAL, EXEMPLARY, OR CONSEQUENTIAL DAMAGES
(INCLUDING, BUT NOT LIMITED TO, PROCUREMENT OF SUBSTITUTE GOODS OR SERVICES;
LOSS OF USE, DATA, OR PROFITS; OR BUSINESS INTERRUPTION) HOWEVER CAUSED AND
ON ANY THEORY OF LIABILITY, WHETHER IN CONTRACT, STRICT LIABILITY, OR TORT
(INCLUDING NEGLIGENCE OR OTHERWISE) ARISING IN ANY WAY OUT OF THE USE OF THIS
SOFTWARE, EVEN IF ADVISED OF THE POSSIBILITY OF SUCH DAMAGE.

*/
#include "IOModule_X20DO6322.hpp"

// Raw Registers
#define JOURNALVARIABLE_X20DO6322_MODULEOK 1
#define JOURNALVARIABLE_X20DO6322_SERIALNUMBER 2
#define JOURNALVARIABLE_X20DO6322_MODULEID 3
#define JOURNALVARIABLE_X20DO6322_HARDWAREVARIANT 4
#define JOURNALVARIABLE_X20DO6322_FIRMWAREVERSION 5
#define JOURNALVARIABLE_X20DO6322_DIGITALOUTPUT01 6
#define JOURNALVARIABLE_X20DO6322_DIGITALOUTPUT02 7
#define JOURNALVARIABLE_X20DO6322_DIGITALOUTPUT03 8
#define JOURNALVARIABLE_X20DO6322_DIGITALOUTPUT04 9
#define JOURNALVARIABLE_X20DO6322_DIGITALOUTPUT05 10
#define JOURNALVARIABLE_X20DO6322_DIGITALOUTPUT06 11
#define JOURNALVARIABLE_X20DO6322_STATUSDIGITALOUTPUT01 12
#define JOURNALVARIABLE_X20DO6322_STATUSDIGITALOUTPUT02 13
#define JOURNALVARIABLE_X20DO6322_STATUSDIGITALOUTPUT03 14
#define JOURNALVARIABLE_X20DO6322_STATUSDIGITALOUTPUT04 15
#define JOURNALVARIABLE_X20DO6322_STATUSDIGITALOUTPUT05 16
#define JOURNALVARIABLE_X20DO6322_STATUSDIGITALOUTPUT06 17

namespace BuRCPP {

	CIOModule_X20DO6322	::CIOModule_X20DO6322 (const std::string & sName, IOMappingX20DO6322_TYP * pMapping)
	: CIOModule (sName), m_pMapping (pMapping)
	{

	}

	CIOModule_X20DO6322::~CIOModule_X20DO6322 ()
	{
	}

	void CIOModule_X20DO6322::onRegisterJournal ()
	{
		registerBoolValue ("ModuleOk", JOURNALVARIABLE_X20DO6322_MODULEOK);
		registerUInt32Value ("SerialNumber", JOURNALVARIABLE_X20DO6322_SERIALNUMBER);
		registerUInt16Value ("ModuleID", JOURNALVARIABLE_X20DO6322_MODULEID);
		registerUInt16Value ("HardwareVariant", JOURNALVARIABLE_X20DO6322_HARDWAREVARIANT);
		registerUInt16Value ("FirmwareVersion", JOURNALVARIABLE_X20DO6322_FIRMWAREVERSION);
		registerBoolValue ("DigitalOutput01", JOURNALVARIABLE_X20DO6322_DIGITALOUTPUT01);
		registerBoolValue ("DigitalOutput02", JOURNALVARIABLE_X20DO6322_DIGITALOUTPUT02);
		registerBoolValue ("DigitalOutput03", JOURNALVARIABLE_X20DO6322_DIGITALOUTPUT03);
		registerBoolValue ("DigitalOutput04", JOURNALVARIABLE_X20DO6322_DIGITALOUTPUT04);
		registerBoolValue ("DigitalOutput05", JOURNALVARIABLE_X20DO6322_DIGITALOUTPUT05);
		registerBoolValue ("DigitalOutput06", JOURNALVARIABLE_X20DO6322_DIGITALOUTPUT06);
		registerBoolValue ("StatusDigitalOutput01", JOURNALVARIABLE_X20DO6322_STATUSDIGITALOUTPUT01);
		registerBoolValue ("StatusDigitalOutput02", JOURNALVARIABLE_X20DO6322_STATUSDIGITALOUTPUT02);
		registerBoolValue ("StatusDigitalOutput03", JOURNALVARIABLE_X20DO6322_STATUSDIGITALOUTPUT03);
		registerBoolValue ("StatusDigitalOutput04", JOURNALVARIABLE_X20DO6322_STATUSDIGITALOUTPUT04);
		registerBoolValue ("StatusDigitalOutput05", JOURNALVARIABLE_X20DO6322_STATUSDIGITALOUTPUT05);
		registerBoolValue ("StatusDigitalOutput06", JOURNALVARIABLE_X20DO6322_STATUSDIGITALOUTPUT06);

	}

	void CIOModule_X20DO6322::onUpdateJournal ()
	{
		setBoolValue (JOURNALVARIABLE_X20DO6322_MODULEOK, m_pMapping->ModuleOk);
		setIntegerValue (JOURNALVARIABLE_X20DO6322_SERIALNUMBER, m_pMapping->SerialNumber);
		setIntegerValue (JOURNALVARIABLE_X20DO6322_MODULEID, m_pMapping->ModuleID);
		setIntegerValue (JOURNALVARIABLE_X20DO6322_HARDWAREVARIANT, m_pMapping->HardwareVariant);
		setIntegerValue (JOURNALVARIABLE_X20DO6322_FIRMWAREVERSION, m_pMapping->FirmwareVersion);
		setBoolValue (JOURNALVARIABLE_X20DO6322_DIGITALOUTPUT01, m_pMapping->DigitalOutput01);
		setBoolValue (JOURNALVARIABLE_X20DO6322_DIGITALOUTPUT02, m_pMapping->DigitalOutput02);
		setBoolValue (JOURNALVARIABLE_X20DO6322_DIGITALOUTPUT03, m_pMapping->DigitalOutput03);
		setBoolValue (JOURNALVARIABLE_X20DO6322_DIGITALOUTPUT04, m_pMapping->DigitalOutput04);
		setBoolValue (JOURNALVARIABLE_X20DO6322_DIGITALOUTPUT05, m_pMapping->DigitalOutput05);
		setBoolValue (JOURNALVARIABLE_X20DO6322_DIGITALOUTPUT06, m_pMapping->DigitalOutput06);
		setBoolValue (JOURNALVARIABLE_X20DO6322_STATUSDIGITALOUTPUT01, m_pMapping->StatusDigitalOutput01);
		setBoolValue (JOURNALVARIABLE_X20DO6322_STATUSDIGITALOUTPUT02, m_pMapping->StatusDigitalOutput02);
		setBoolValue (JOURNALVARIABLE_X20DO6322_STATUSDIGITALOUTPUT03, m_pMapping->StatusDigitalOutput03);
		setBoolValue (JOURNALVARIABLE_X20DO6322_STATUSDIGITALOUTPUT04, m_pMapping->StatusDigitalOutput04);
		setBoolValue (JOURNALVARIABLE_X20DO6322_STATUSDIGITALOUTPUT05, m_pMapping->StatusDigitalOutput05);
		setBoolValue (JOURNALVARIABLE_X20DO6322_STATUSDIGITALOUTPUT06, m_pMapping->StatusDigitalOutput06);
	}

	bool CIOModule_X20DO6322::isActive ()
	{
		return m_pMapping->ModuleOk != 0;
	}

	uint32_t CIOModule_X20DO6322::getSerialNumber ()
	{
		return m_pMapping->SerialNumber;
	}

	uint16_t CIOModule_X20DO6322::getModuleID ()
	{
		return m_pMapping->ModuleID;
	}

	uint16_t CIOModule_X20DO6322::getHardwareVariant ()
	{
		return m_pMapping->HardwareVariant;
	}

	uint16_t CIOModule_X20DO6322::getFirmwareVersion ()
	{
		return m_pMapping->FirmwareVersion;
	}

	void CIOModule_X20DO6322::setOutput (uint32_t nChannelNo, bool nValue)
	{
		switch (nChannelNo)
		{
			case 1:
				m_pMapping->DigitalOutput01 = nValue;
				break;

			case 2:
				m_pMapping->DigitalOutput02 = nValue;
				break;

			case 3:
				m_pMapping->DigitalOutput03 = nValue;
				break;

			case 4:
				m_pMapping->DigitalOutput04 = nValue;
				break;

			case 5:
				m_pMapping->DigitalOutput05 = nValue;
				break;

			case 6:
				m_pMapping->DigitalOutput06 = nValue;
				break;
			default:
				throw CException (eErrorCode::INVALIDCHANNELNUMBER, "invalid channel number: " + std::to_string (nChannelNo));
		}

	}

	bool CIOModule_X20DO6322::getOutput (uint32_t nChannelNo)
	{
		switch (nChannelNo)
		{
			case 1:
				return m_pMapping->DigitalOutput01;

			case 2:
				return m_pMapping->DigitalOutput02;

			case 3:
				return m_pMapping->DigitalOutput03;

			case 4:
				return m_pMapping->DigitalOutput04;

			case 5:
				return m_pMapping->DigitalOutput05;

			case 6:
				return m_pMapping->DigitalOutput06;

			default:
				throw CException (eErrorCode::INVALIDCHANNELNUMBER, "invalid channel number: " + std::to_string (nChannelNo));
		}

	}

	uint16_t CIOModule_X20DO6322::getIOStatus (uint32_t nChannelNo)
	{
		/*status IDs: 0 = no error, 1 = short circuit or overload, or channel switched on and missing I/O power supply,
		or channel switched off and external voltage applied on channel*/

		switch (nChannelNo)
		{
			case 1: return m_pMapping->StatusDigitalOutput01;
			case 2: return m_pMapping->StatusDigitalOutput02;
			case 3: return m_pMapping->StatusDigitalOutput03;
			case 4: return m_pMapping->StatusDigitalOutput04;
			case 5: return m_pMapping->StatusDigitalOutput05;
			case 6: return m_pMapping->StatusDigitalOutput06;
			default:
				throw CException (eErrorCode::INVALIDCHANNELNUMBER, "invalid channel number: " + std::to_string (nChannelNo));
		}
	}

}
```

#### IOModule_X20AO4622.hpp
```cpp
/*++

Copyright (C) 2024 Institute for Machine Tools and Industrial Management
TUM School of Engineering and Design
Technical University of Munich

All rights reserved.

Redistribution and use in source and binary forms, with or without
modification, are permitted provided that the following conditions are met:
	* Redistributions of source code must retain the above copyright
	  notice, this list of conditions and the following disclaimer.
	* Redistributions in binary form must reproduce the above copyright
	  notice, this list of conditions and the following disclaimer in the
	  documentation and/or other materials provided with the distribution.
	* Neither the name of the Technical University of Munich nor the
	  names of its contributors may be used to endorse or promote products
	  derived from this software without specific prior written permission.

THIS SOFTWARE IS PROVIDED BY THE COPYRIGHT HOLDERS AND CONTRIBUTORS "AS IS" AND
ANY EXPRESS OR IMPLIED WARRANTIES, INCLUDING, BUT NOT LIMITED TO, THE IMPLIED
WARRANTIES OF MERCHANTABILITY AND FITNESS FOR A PARTICULAR PURPOSE ARE
DISCLAIMED. IN NO EVENT SHALL TECHNICAL UNIVERSITY OF MUNICH BE LIABLE FOR ANY
DIRECT, INDIRECT, INCIDENTAL, SPECIAL, EXEMPLARY, OR CONSEQUENTIAL DAMAGES
(INCLUDING, BUT NOT LIMITED TO, PROCUREMENT OF SUBSTITUTE GOODS OR SERVICES;
LOSS OF USE, DATA, OR PROFITS; OR BUSINESS INTERRUPTION) HOWEVER CAUSED AND
ON ANY THEORY OF LIABILITY, WHETHER IN CONTRACT, STRICT LIABILITY, OR TORT
(INCLUDING NEGLIGENCE OR OTHERWISE) ARISING IN ANY WAY OUT OF THE USE OF THIS
SOFTWARE, EVEN IF ADVISED OF THE POSSIBILITY OF SUCH DAMAGE.

*/

#ifndef __IOMODULE_X20AO4622_HPP
#define __IOMODULE_X20AO4622_HPP

#include "../Framework/Framework.hpp"

namespace BuRCPP {

	enum class eIOChannelType_X20AO4622 : uint32_t {
		mtUnknown = 0,
		mtVoltage10V = 1,
		mtCurrent0to20mA = 2,
		mtCurrent4to20mA = 3
	};

	class CIOModule_X20AO4622 : public CIOModule {
		protected:
		IOMappingX20AO4622_TYP * m_pMapping;
		std::array<eIOChannelType_X20AO4622, 4>  m_ChannelTypes;
		std::array<int16_t,4> m_nLowerLimit;
		std::array<int16_t,4> m_nUpperLimit;

		public:
		CIOModule_X20AO4622 (const std::string & sName, IOMappingX20AO4622_TYP * pMapping);
		virtual ~CIOModule_X20AO4622 ();

		bool isActive () override;

		bool setRange(uint32_t nChannelNo, uint16_t nLower, uint16_t nUpper);

		uint32_t getSerialNumber () override;
		uint16_t getModuleID () override;
		uint16_t getHardwareVariant () override;
		uint16_t getFirmwareVersion () override;
		eIOChannelType_X20AO4622 getChannelType (uint32_t nChannelNo);
		bool setChannelType (uint32_t nChannelNo, eIOChannelType_X20AO4622 eChannelTypes);

		int16_t getRawValue (uint32_t nChannelNo);
		double getRawValueNormalizedZeroToOne (uint32_t nChannelNo);
		double getOutputVoltageInVolt (uint32_t nChannelNo);
		double getOutputCurrentInAmpere (uint32_t nChannelNo);

		void setRawValueNormalizedZeroToOne (uint32_t nChannelNo, double dRawValueNormalizedZeroToOne);
		void setOutputVoltageInVolt (uint32_t nChannelNo, double dOutputVoltageInVolt);
		void setOutputCurrentInAmpere (uint32_t nChannelNo, double dOutputCurrentInAmpere);

		virtual void onRegisterJournal () override;
		virtual void onUpdateJournal () override;

	};

}

#endif //__IOMODULE_X20AO4622_HPP
```

#### IOModule_X20AO4622.cpp
```cpp
/*++

Copyright (C) 2024 Institute for Machine Tools and Industrial Management
TUM School of Engineering and Design
Technical University of Munich

All rights reserved.

Redistribution and use in source and binary forms, with or without
modification, are permitted provided that the following conditions are met:
	* Redistributions of source code must retain the above copyright
	  notice, this list of conditions and the following disclaimer.
	* Redistributions in binary form must reproduce the above copyright
	  notice, this list of conditions and the following disclaimer in the
	  documentation and/or other materials provided with the distribution.
	* Neither the name of the Technical University of Munich nor the
	  names of its contributors may be used to endorse or promote products
	  derived from this software without specific prior written permission.

THIS SOFTWARE IS PROVIDED BY THE COPYRIGHT HOLDERS AND CONTRIBUTORS "AS IS" AND
ANY EXPRESS OR IMPLIED WARRANTIES, INCLUDING, BUT NOT LIMITED TO, THE IMPLIED
WARRANTIES OF MERCHANTABILITY AND FITNESS FOR A PARTICULAR PURPOSE ARE
DISCLAIMED. IN NO EVENT SHALL TECHNICAL UNIVERSITY OF MUNICH BE LIABLE FOR ANY
DIRECT, INDIRECT, INCIDENTAL, SPECIAL, EXEMPLARY, OR CONSEQUENTIAL DAMAGES
(INCLUDING, BUT NOT LIMITED TO, PROCUREMENT OF SUBSTITUTE GOODS OR SERVICES;
LOSS OF USE, DATA, OR PROFITS; OR BUSINESS INTERRUPTION) HOWEVER CAUSED AND
ON ANY THEORY OF LIABILITY, WHETHER IN CONTRACT, STRICT LIABILITY, OR TORT
(INCLUDING NEGLIGENCE OR OTHERWISE) ARISING IN ANY WAY OUT OF THE USE OF THIS
SOFTWARE, EVEN IF ADVISED OF THE POSSIBILITY OF SUCH DAMAGE.

*/
#include "IOModule_X20AO4622.hpp"

// Raw Registers
#define JOURNALVARIABLE_X20AO4622_MODULEOK 1
#define JOURNALVARIABLE_X20AO4622_SERIALNUMBER 3
#define JOURNALVARIABLE_X20AO4622_MODULEID 4
#define JOURNALVARIABLE_X20AO4622_HARDWAREVARIANT 5
#define JOURNALVARIABLE_X20AO4622_FIRMWAREVERSION 6
#define JOURNALVARIABLE_X20AO4622_ANALOGOUTPUT01 7
#define JOURNALVARIABLE_X20AO4622_ANALOGOUTPUT02 8
#define JOURNALVARIABLE_X20AO4622_ANALOGOUTPUT03 9
#define JOURNALVARIABLE_X20AO4622_ANALOGOUTPUT04 10

// Derived Values
#define JOURNALVARIABLE_X20AO4622_OUTPUTVOLTAGE01 1001
#define JOURNALVARIABLE_X20AO4622_OUTPUTVOLTAGE02 1002
#define JOURNALVARIABLE_X20AO4622_OUTPUTVOLTAGE03 1003
#define JOURNALVARIABLE_X20AO4622_OUTPUTVOLTAGE04 1004
#define JOURNALVARIABLE_X20AO4622_OUTPUTCURRENTINAMPERE01 1005
#define JOURNALVARIABLE_X20AO4622_OUTPUTCURRENTINAMPERE02 1006
#define JOURNALVARIABLE_X20AO4622_OUTPUTCURRENTINAMPERE03 1007
#define JOURNALVARIABLE_X20AO4622_OUTPUTCURRENTINAMPERE04 1008

namespace BuRCPP {

	CIOModule_X20AO4622	::CIOModule_X20AO4622 (const std::string & sName, IOMappingX20AO4622_TYP * pMapping)
		: CIOModule (sName), m_pMapping (pMapping)
	{
		for (auto &channelType:m_ChannelTypes)
			channelType = eIOChannelType_X20AO4622::mtVoltage10V;

		for (auto &LowerLimits:m_nLowerLimit)
			LowerLimits = -32767;

		for (auto &UpperLimits:m_nUpperLimit)
			UpperLimits = 32766;

	}

	CIOModule_X20AO4622::~CIOModule_X20AO4622 ()
	{
	}

	void CIOModule_X20AO4622::onRegisterJournal ()
	{
		registerBoolValue ("ModuleOk", JOURNALVARIABLE_X20AO4622_MODULEOK);
		registerUInt32Value ("SerialNumber", JOURNALVARIABLE_X20AO4622_SERIALNUMBER);
		registerUInt16Value ("ModuleID", JOURNALVARIABLE_X20AO4622_MODULEID);
		registerUInt16Value ("HardwareVariant", JOURNALVARIABLE_X20AO4622_HARDWAREVARIANT);
		registerUInt16Value ("FirmwareVersion", JOURNALVARIABLE_X20AO4622_FIRMWAREVERSION);
		registerInt16Value ("AnalogOutput01", JOURNALVARIABLE_X20AO4622_ANALOGOUTPUT01);
		registerInt16Value ("AnalogOutput02", JOURNALVARIABLE_X20AO4622_ANALOGOUTPUT02);
		registerInt16Value ("AnalogOutput03", JOURNALVARIABLE_X20AO4622_ANALOGOUTPUT03);
		registerInt16Value ("AnalogOutput04", JOURNALVARIABLE_X20AO4622_ANALOGOUTPUT04);

		switch (getChannelType (1)) {
			case eIOChannelType_X20AO4622::mtVoltage10V:
				registerDoubleValue ("OutputVoltage01", JOURNALVARIABLE_X20AO4622_OUTPUTVOLTAGE01, -10.0, 10.0, 65536);
				break;

			case eIOChannelType_X20AO4622::mtCurrent0to20mA:
				registerDoubleValue ("OutputCurrentInAmpere01", JOURNALVARIABLE_X20AO4622_OUTPUTCURRENTINAMPERE01, 0.000, 0.020, 65536);
				break;

			case eIOChannelType_X20AO4622::mtCurrent4to20mA:
				registerDoubleValue ("OutputCurrentInAmpere01", JOURNALVARIABLE_X20AO4622_OUTPUTCURRENTINAMPERE01, 0.004, 0.020, 65536);
				break;
		}

		switch (getChannelType (2)) {
			case eIOChannelType_X20AO4622::mtVoltage10V:
				registerDoubleValue ("OutputVoltage02", JOURNALVARIABLE_X20AO4622_OUTPUTVOLTAGE02, -10.0, 10.0, 65536);
				break;

			case eIOChannelType_X20AO4622::mtCurrent0to20mA:
				registerDoubleValue ("OutputCurrentInAmpere02", JOURNALVARIABLE_X20AO4622_OUTPUTCURRENTINAMPERE02, 0.000, 0.020, 65536);
				break;

			case eIOChannelType_X20AO4622::mtCurrent4to20mA:
				registerDoubleValue ("OutputCurrentInAmpere02", JOURNALVARIABLE_X20AO4622_OUTPUTCURRENTINAMPERE02, 0.004, 0.020, 65536);
				break;
		}

		switch (getChannelType (3)) {
			case eIOChannelType_X20AO4622::mtVoltage10V:
				registerDoubleValue ("OutputVoltage03", JOURNALVARIABLE_X20AO4622_OUTPUTVOLTAGE03, -10.0, 10.0, 65536);
				break;

			case eIOChannelType_X20AO4622::mtCurrent0to20mA:
				registerDoubleValue ("OutputCurrentInAmpere03", JOURNALVARIABLE_X20AO4622_OUTPUTCURRENTINAMPERE03, 0.000, 0.020, 65536);
				break;

			case eIOChannelType_X20AO4622::mtCurrent4to20mA:
				registerDoubleValue ("OutputCurrentInAmpere03", JOURNALVARIABLE_X20AO4622_OUTPUTCURRENTINAMPERE03, 0.004, 0.020, 65536);
				break;
		}

		switch (getChannelType (4)) {
			case eIOChannelType_X20AO4622::mtVoltage10V:
				registerDoubleValue ("OutputVoltage04", JOURNALVARIABLE_X20AO4622_OUTPUTVOLTAGE04, -10.0, 10.0, 65536);
				break;

			case eIOChannelType_X20AO4622::mtCurrent0to20mA:
				registerDoubleValue ("OutputCurrentInAmpere04", JOURNALVARIABLE_X20AO4622_OUTPUTCURRENTINAMPERE04, 0.000, 0.020, 65536);
				break;

			case eIOChannelType_X20AO4622::mtCurrent4to20mA:
				registerDoubleValue ("OutputCurrentInAmpere04", JOURNALVARIABLE_X20AO4622_OUTPUTCURRENTINAMPERE04, 0.004, 0.020, 65536);
				break;
		}
	}

	void CIOModule_X20AO4622::onUpdateJournal ()
	{
		setBoolValue (JOURNALVARIABLE_X20AO4622_MODULEOK, m_pMapping->ModuleOk);
		setIntegerValue (JOURNALVARIABLE_X20AO4622_SERIALNUMBER, m_pMapping->SerialNumber);
		setIntegerValue (JOURNALVARIABLE_X20AO4622_MODULEID, m_pMapping->ModuleID);
		setIntegerValue (JOURNALVARIABLE_X20AO4622_HARDWAREVARIANT, m_pMapping->HardwareVariant);
		setIntegerValue (JOURNALVARIABLE_X20AO4622_FIRMWAREVERSION, m_pMapping->FirmwareVersion);
		setIntegerValue (JOURNALVARIABLE_X20AO4622_ANALOGOUTPUT01, m_pMapping->AnalogOutput01);
		setIntegerValue (JOURNALVARIABLE_X20AO4622_ANALOGOUTPUT02, m_pMapping->AnalogOutput02);
		setIntegerValue (JOURNALVARIABLE_X20AO4622_ANALOGOUTPUT03, m_pMapping->AnalogOutput03);
		setIntegerValue (JOURNALVARIABLE_X20AO4622_ANALOGOUTPUT03, m_pMapping->AnalogOutput04);

		for (int index = 0; index < 4; index++)
		{
			uint32_t nChannelNo = index + 1;
			switch (getChannelType (nChannelNo)) {

				case eIOChannelType_X20AO4622::mtVoltage10V:

					setDoubleValue (JOURNALVARIABLE_X20AO4622_OUTPUTVOLTAGE01 + index, getOutputVoltageInVolt (nChannelNo));
					break;

				case eIOChannelType_X20AO4622::mtCurrent0to20mA:
				case eIOChannelType_X20AO4622::mtCurrent4to20mA:
					setDoubleValue (JOURNALVARIABLE_X20AO4622_OUTPUTCURRENTINAMPERE01 + index, getOutputCurrentInAmpere (nChannelNo));
					break;
			}
		}
	}

	bool CIOModule_X20AO4622::isActive ()
	{
		return m_pMapping->ModuleOk != 0;
	}

	uint32_t CIOModule_X20AO4622::getSerialNumber ()
	{
		return m_pMapping->SerialNumber;
	}

	uint16_t CIOModule_X20AO4622::getModuleID ()
	{
		return m_pMapping->ModuleID;
	}

	uint16_t CIOModule_X20AO4622::getHardwareVariant ()
	{
		return m_pMapping->HardwareVariant;
	}

	uint16_t CIOModule_X20AO4622::getFirmwareVersion ()
	{
		return m_pMapping->FirmwareVersion;
	}

	int16_t CIOModule_X20AO4622::getRawValue (uint32_t nChannelNo)
	{

		switch (nChannelNo) {
			case 1: return m_pMapping->AnalogOutput01;
			case 2: return m_pMapping->AnalogOutput02;
			case 3: return m_pMapping->AnalogOutput03;
			case 4: return m_pMapping->AnalogOutput04;
			default:
				throw CException (eErrorCode::INVALIDCHANNELNUMBER, "invalid channel number: " + std::to_string (nChannelNo));
		}
	}

	double CIOModule_X20AO4622::getRawValueNormalizedZeroToOne (uint32_t nChannelNo)
	{
		if (nChannelNo > 0 && nChannelNo < 5)
		{
			int32_t rawValue = getRawValue (nChannelNo);
			int32_t nRange = m_nUpperLimit[nChannelNo -1] - m_nLowerLimit[nChannelNo -1];
			return (double) (rawValue - (int32_t) m_nLowerLimit[nChannelNo -1]) / (double) nRange;
		}
		else
		{
			throw CException (eErrorCode::INVALIDCHANNELNUMBER, "invalid channel number: " + std::to_string (nChannelNo));
		}
	}

	double CIOModule_X20AO4622::getOutputVoltageInVolt (uint32_t nChannelNo)
	{
		switch (getChannelType (nChannelNo)) {
			case eIOChannelType_X20AO4622::mtVoltage10V:
				return (getRawValueNormalizedZeroToOne (nChannelNo) - 0.5) * 20.0;
			default:
				throw CException (eErrorCode::NOVOLTAGEMODULE, "IO module does not measure voltage: " + m_sName );
		}

	}

	double CIOModule_X20AO4622::getOutputCurrentInAmpere (uint32_t nChannelNo)
	{
		switch (getChannelType (nChannelNo)) {
			case eIOChannelType_X20AO4622::mtCurrent0to20mA:
				return (getRawValueNormalizedZeroToOne (nChannelNo)) * 0.020;
			case eIOChannelType_X20AO4622::mtCurrent4to20mA:
				return (getRawValueNormalizedZeroToOne (nChannelNo)) * 0.016 + 0.004;
			default:
				throw CException (eErrorCode::NOCURRENTMODULE, "IO module does not measure current: " + m_sName );
		}

	}

	bool CIOModule_X20AO4622::setRange(uint32_t nChannelNo, uint16_t nLower, uint16_t nUpper)
	{
		if (nChannelNo > 0 && nChannelNo < 5)
		{
			m_nLowerLimit[nChannelNo - 1] = nLower;
			m_nUpperLimit[nChannelNo - 1] = nUpper;
			return true;
		}
		else
		{
			return false;
		}
	}

	eIOChannelType_X20AO4622 CIOModule_X20AO4622::getChannelType (uint32_t nChannelNo)
	{
		if ((nChannelNo >= 1) && (nChannelNo <= 4))
		{
			return m_ChannelTypes[nChannelNo - 1];
		}
		else
			return eIOChannelType_X20AO4622::mtUnknown;
	}

	bool CIOModule_X20AO4622::setChannelType (uint32_t nChannelNo, eIOChannelType_X20AO4622 eChannelTypes)
	{
		if ((nChannelNo >= 1) && (nChannelNo <= 4))
		{
			switch (eChannelTypes) {
				case eIOChannelType_X20AO4622::mtVoltage10V:
					setRange(nChannelNo, -32768 , 32767);
					break;
				case eIOChannelType_X20AO4622::mtCurrent0to20mA:
					setRange(nChannelNo, 0, 32767);
					break;
				case eIOChannelType_X20AO4622::mtCurrent4to20mA:
					setRange(nChannelNo, -8192 , 32767);
					break;
				default:
					throw CException (eErrorCode::INVALIDCHANNELTYPE, "invalid channel type");
			}
			m_ChannelTypes[nChannelNo - 1] = eChannelTypes;
			return true;
		}
		else
		{
			throw CException (eErrorCode::INVALIDCHANNELNUMBER, "invalid channel number: " + std::to_string (nChannelNo));
		}

	}

	void CIOModule_X20AO4622::setRawValueNormalizedZeroToOne (uint32_t nChannelNo, double dRawValueNormalizedZeroToOne)
	{
		if ( 0.0<= dRawValueNormalizedZeroToOne <= 1.0)
		{
			int32_t rawValue = m_nLowerLimit[nChannelNo -1] + (m_nUpperLimit[nChannelNo -1] - m_nLowerLimit[nChannelNo -1])*dRawValueNormalizedZeroToOne;

			switch (nChannelNo)
			{
				case 1:
					m_pMapping->AnalogOutput01 = rawValue;
					return;

				case 2:
					m_pMapping->AnalogOutput02 = rawValue;
					return;

				case 3:
					m_pMapping->AnalogOutput03 = rawValue;
					return;

				case 4:
					m_pMapping->AnalogOutput04 = rawValue;
					return;
				default:
					throw CException (eErrorCode::INVALIDCHANNELNUMBER, "invalid channel number: " + std::to_string (nChannelNo));
			}
		}
		else
		{
			throw CException (eErrorCode::INVALIDCHANNELVALUE, "invalid channel value: " + std::to_string (dRawValueNormalizedZeroToOne));
		}
	}

	void CIOModule_X20AO4622::setOutputVoltageInVolt (uint32_t nChannelNo, double dOutputVoltageInVolt)
	{
		if(getChannelType(nChannelNo) == eIOChannelType_X20AO4622::mtVoltage10V)
		{
			if ( -10.0 <= dOutputVoltageInVolt <= 10.0)
			{
				double dNormalizedValueZeroToOne = (dOutputVoltageInVolt+10.0)/20.0;
				setRawValueNormalizedZeroToOne(nChannelNo,dNormalizedValueZeroToOne);
				return;
			}
			else
			{
				throw CException (eErrorCode::INVALIDCHANNELVALUE, "invalid channel value: " + std::to_string (dOutputVoltageInVolt));
			}

		}
		else
		{
			throw CException (eErrorCode::NOVOLTAGEMODULE, "IO module does not measure voltage: " + m_sName );
		}

	}

	void CIOModule_X20AO4622::setOutputCurrentInAmpere (uint32_t nChannelNo, double dOutputCurrentInAmpere)
	{
		switch (getChannelType (nChannelNo)) {
			case eIOChannelType_X20AO4622::mtCurrent0to20mA:
				if ( 0.0 <= dOutputCurrentInAmpere <= 0.02)
				{
					double dNormalizedValueZeroToOne = (dOutputCurrentInAmpere)/0.02;
					setRawValueNormalizedZeroToOne(nChannelNo,dNormalizedValueZeroToOne);
					return;
				}
				else
				{
					throw CException (eErrorCode::INVALIDCHANNELVALUE, "invalid channel value: " + std::to_string (dOutputCurrentInAmpere));
				}
				return;
			case eIOChannelType_X20AO4622::mtCurrent4to20mA:
				if ( 0.004 <= dOutputCurrentInAmpere <= 0.02)
				{
					double dNormalizedValueZeroToOne = (dOutputCurrentInAmpere-0.004)/0.016;
					setRawValueNormalizedZeroToOne(nChannelNo,dNormalizedValueZeroToOne);
					return;
				}
				else
				{
					throw CException (eErrorCode::INVALIDCHANNELVALUE, "invalid channel value: " + std::to_string (dOutputCurrentInAmpere));
				}
				return;
			default:
				throw CException (eErrorCode::NOCURRENTMODULE, "IO module does not measure current: " + m_sName );
		}
	}

}
```
